// TIA Portal V20 export
// export: Created 2025-12-01T14:56:47.7137702Z, ExportSetting None, DisplayName Totally Integrated Automation Portal, DisplayVersion V20 Update 3, DisplayName TIA Portal Openness, DisplayVersion V20 Update 3, DisplayName TIA Portal Version Control Interface, DisplayVersion V20 Update 3, DisplayName STEP 7 Professional, DisplayVersion V20 Update 3, DisplayName STEP 7 Safety, DisplayVersion V20 Update 2, DisplayName WinCC Basic/Comfort/Advanced, DisplayVersion V20 Update 3, DisplayName WinCC Professional, DisplayVersion V20 Update 3, DisplayName WinCC Unified, DisplayVersion V20 Update 3
FUNCTION_BLOCK "FB350_Apilador_DesApilador_Paletas"   // FB350, LAD
TITLE = Control del Ramal de Salidas
{ S7_Optimized_Access := 'FALSE' }
AUTHOR : MAQUINA
NAME : 20181114
VERSION : 3.5
// Dani Palacios: Modificación octubre 2017 para poder desabilitar la maquina con un bit (por ejemplo en la puesta a punto si no esta montada o en el simulador)
// La modificación esta sin probar y es todo lo relativo a la variable Maquina_Desabilitada
// (bloqueo evolución desde etapa 0, bloqueo activación salidas en etapa 0 , fin vi sin mirar detectores y activación posición de reposo sin mirar detectores y variabkles de fin de movimiento).
// ES RESPONSABILIDAD DEL QUE DESABILITA LA MAQUINA QUE ESTA ESTE EN UNA POSICION QUE PERMITA EL MOVIMIENTO DE LAS CARGAS A TRAVES DE ELLA
// stored: AutoNumber false, SetENOAutomatically false
   VAR_INPUT
      Maquina : UInt;   // Numero de Maquina (Mesa)
      Error_Tx : Bool;   // Error en el Tx
      EnTension : Bool;   // Existe Tension en la Mesa
      MAQx_Desabilitada : Bool;   // Config MAQ. >>> DesHabilitada
      MAQx_ReposoDW : Bool;   // Config MAQ. >>> Pos. Reposo Abajo
      Termico_Elevacion : Bool;   // Termico de la Elevacion
      Termico_HorqDch : Bool;   // Termico de la Horquilla Derecha
      Termico_HorqIzq : Bool;   // Termico de la horquilla Izquierda
      pHsMx : Bool;   // pHs de la Mesa
      EnMovimiento_Tx : Bool;   // En Movimiento Tx
      pHs_LlenoApilador : Bool;   // Lleno el Apilador
      pHs_ConCargaApilador : Bool;   // ConCarga Apilador
      EM_UP : Bool;   // Emergencia Arriba del Apilador
      EM_DW : Bool;   // Emergencia Abajo del Apilador
      Pos_Dw : Bool;   // Posición Baja del Apilador
      Pos_Mid : Bool;   // Posición Media del Apilador
      Pos_Up : Bool;   // Posición Alta del Apilador
      Horq1_Der_Recogida : Bool;
      Horq2_Der_Recogida : Bool;
      Horq1_Izq_Recogida : Bool;
      Horq2_Izq_Recogida : Bool;
      Horq1_Der_Extendida : Bool;
      Horq2_Der_Extendida : Bool;
      Horq1_Izq_Extendida : Bool;
      Horq2_Izq_Extendida : Bool;
      EnMovimiento_Elevacion : Bool;   // En Movineto la Elevacion
      EnMovimiento_Horquillado : Bool;   // En Movimiento el Hoquillado
      PasarReposo_Apilador : Bool;   // Pasar a Reposo >>> Interlock Maquina
      CogerPila_Apilador : Bool;   // Coger la Pila >>> Interlock Maquina
      DispensarPaleta_Apilador : Bool;   // Dispensar Paleta >>> Interlock Maquina
      DispensarpPila_Apilador : Bool;   // Dispensar Pila >>> Interlock Maquina
      V_TIM_EstabilidadMov : Time := T#200MS;   // TIM de Estabilidad de los Mov.
      V_TOut_Elevacion : Int := 10000;   // TimeOut del Mov. de Elevacion
      V_TOut_Horquillado : Int := 3000;   // TimeOut del Mov. de Horquillado
   END_VAR
   VAR_OUTPUT
      Quieto_Apilador : Bool;   // Quieto >>> Interlock Maquina
      FinMovimiento_Apilador : Bool;   // Fin Movimiento >>> Interlock Maquina
   END_VAR
   VAR_IN_OUT
      StatusLleno_Apilador : Bool;   // Status Lleno >>> Interlock Maquina
      StatusSemiLleno_Apilador : Bool;   // Status SemiLleno >>> Interlock Maquina
      StatusVacio_Apilador : Bool;   // Status Vacio >>> Interlock Maquina
   END_VAR
   VAR
      Ap_ET00 : Bool;
      Ap_ET100 : Bool;
      Ap_ET101 : Bool;
      Ap_ET102 : Bool;
      Ap_ET103 : Bool;
      Ap_ET104 : Bool;
      Ap_ET105 : Bool;
      Ap_ET106 : Bool;
      Ap_ET107 : Bool;
      Ap_ET108 : Bool;
      Ap_ET109 : Bool;
      Ap_ET11 : Bool;
      Ap_ET12 : Bool;
      Ap_ET13 : Bool;
      Ap_ET14 : Bool;
      Ap_ET15 : Bool;
      Ap_ET16 : Bool;
      Ap_ET21 : Bool;
      Ap_ET22 : Bool;
      Ap_ET23 : Bool;
      Ap_ET24 : Bool;
      Ap_ET31 : Bool;
      Ap_ET32 : Bool;
      Ap_ET41 : Bool;
      Ap_ET42 : Bool;
      Ap_ET43 : Bool;
      Ap_ET44 : Bool;
      Ap_ET50 : Bool;
      Ap_ET51 : Bool;
      PosicionConocida : Bool;   // Interna >> Posicion Conocida
      Apilador_Lleno : Bool;   // Interna >> Lleno el Apilador
      HorquillasRecogidas : Bool;   // Carga Suelta en el Apilador
      HorquillasExtendidas : Bool;   // Carga Cogida en el Apilador
      STAT_FinMovimiento : Bool;   // Interna >> Fin Movimitnto del Apilador
      STAT_Quieto : Bool;   // Interna >> Quieto el Apilador
      CambioDir_SubidaBajada : Bool;   // Interna >> Cambio de Dir. Subida o Bajada
      MA_Ir_Up : Bool;   // ???
      MA_Ir_Dw : Bool;   // ???
      MA_Ir_Mid_Bajando : Bool;   // ???
      MA_Ir_Mid_Subiendo : Bool;   // ???
      MA_DejarCarga : Bool;   // ???
      MA_CogerCarga : Bool;   // ???
      TIM_EstabilidadMov { S7_SetPoint := 'True'} : TON_TIME;
      TMP_EnTension { S7_SetPoint := 'True'} : "FB910_CNT_UHS";
      TOut_Elevacion { S7_SetPoint := 'True'} : "FB910_CNT_UHS";
      TOut_Horquillado { S7_SetPoint := 'True'} : "FB910_CNT_UHS";
      Manual : "MoviManualMaquina_DesApilador";
   END_VAR
   VAR_TEMP
      EstadoZona : "EstadoZona";   // Estado de Zona de la Mesa
      EstadoMAQ : "EstadoMaquina_ApiladorDesapilador";   // Estado del Vehiculo Inteliguente de la Maquina
      Aux_ET00 : Bool;
   END_VAR
   VAR_TEMP   // added for the SCL form of the ladder/FBD networks
      _w1 : Bool;
   END_VAR
BEGIN

REGION Network 1: INICIALIZAR - Recoger las Variables de Estado de la Maquina
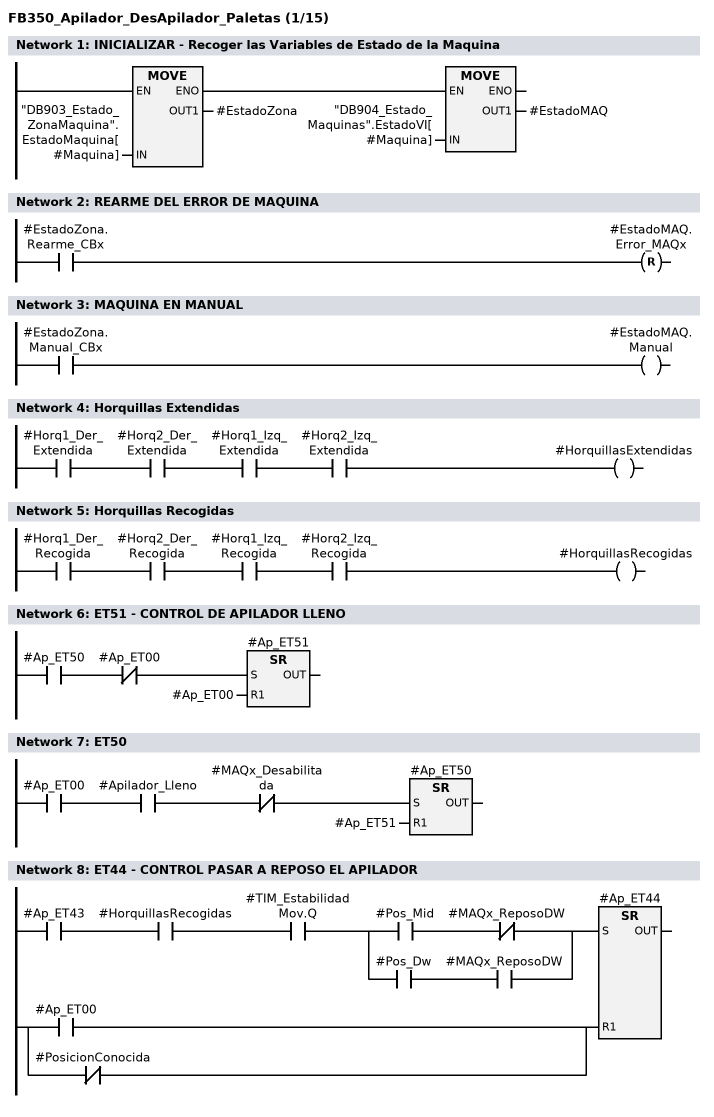
   RUNG wire#powerrail
      Move(in := "DB903_Estado_ZonaMaquina".EstadoMaquina[#Maquina], out1 => #EstadoZona)
      Move(in := "DB904_Estado_Maquinas".EstadoVI[#Maquina], out1 => #EstadoMAQ)
   END_RUNG
   // the same network as SCL:
   #EstadoZona := "DB903_Estado_ZonaMaquina".EstadoMaquina[#Maquina];
   #EstadoMAQ := "DB904_Estado_Maquinas".EstadoVI[#Maquina];
END_REGION

REGION Network 2: REARME DEL ERROR DE MAQUINA
   RUNG wire#powerrail
      Contact( #EstadoZona.Rearme_CBx )
      R_Coil( #EstadoMAQ.Error_MAQx )
   END_RUNG
   // the same network as SCL:
   IF #EstadoZona.Rearme_CBx THEN #EstadoMAQ.Error_MAQx := FALSE; END_IF;
END_REGION

REGION Network 3: MAQUINA EN MANUAL
   RUNG wire#powerrail
      Contact( #EstadoZona.Manual_CBx )
      Coil( #EstadoMAQ.Manual )
   END_RUNG
   // the same network as SCL:
   #EstadoMAQ.Manual := #EstadoZona.Manual_CBx;
END_REGION

REGION Network 4: Horquillas Extendidas
   RUNG wire#powerrail
      Contact( #Horq1_Der_Extendida )
      Contact( #Horq2_Der_Extendida )
      Contact( #Horq1_Izq_Extendida )
      Contact( #Horq2_Izq_Extendida )
      Coil( #HorquillasExtendidas )
   END_RUNG
   // the same network as SCL:
   #HorquillasExtendidas := #Horq1_Der_Extendida AND #Horq2_Der_Extendida AND #Horq1_Izq_Extendida AND #Horq2_Izq_Extendida;
END_REGION

REGION Network 5: Horquillas Recogidas
   RUNG wire#powerrail
      Contact( #Horq1_Der_Recogida )
      Contact( #Horq2_Der_Recogida )
      Contact( #Horq1_Izq_Recogida )
      Contact( #Horq2_Izq_Recogida )
      Coil( #HorquillasRecogidas )
   END_RUNG
   // the same network as SCL:
   #HorquillasRecogidas := #Horq1_Der_Recogida AND #Horq2_Der_Recogida AND #Horq1_Izq_Recogida AND #Horq2_Izq_Recogida;
END_REGION

REGION Network 6: ET51 - CONTROL DE APILADOR LLENO
   RUNG wire#powerrail
      Contact( #Ap_ET50 )
      I_Contact( #Ap_ET00 )
      S_SR(operand := #Ap_ET51, r1 := #Ap_ET00)
   END_RUNG
   // the same network as SCL:
   IF #Ap_ET50 AND NOT #Ap_ET00 THEN
       #Ap_ET51 := TRUE;   // SR flip-flop
   END_IF;
   IF #Ap_ET00 THEN #Ap_ET51 := FALSE; END_IF;
END_REGION

REGION Network 7: ET50
   RUNG wire#powerrail
      Contact( #Ap_ET00 )
      Contact( #Apilador_Lleno )
      I_Contact( #MAQx_Desabilitada )
      S_SR(operand := #Ap_ET50, r1 := #Ap_ET51)
   END_RUNG
   // the same network as SCL:
   IF #Ap_ET00 AND #Apilador_Lleno AND NOT #MAQx_Desabilitada THEN
       #Ap_ET50 := TRUE;   // SR flip-flop
   END_IF;
   IF #Ap_ET51 THEN #Ap_ET50 := FALSE; END_IF;
END_REGION

REGION Network 8: ET44 - CONTROL PASAR A REPOSO EL APILADOR
   RUNG wire#powerrail
      Contact( #Ap_ET43 )
      Contact( #HorquillasRecogidas )
      Contact( #TIM_EstabilidadMov.Q )
      wire#w1
      Contact( #Pos_Mid )
      I_Contact( #MAQx_ReposoDW )
      wire#w2
      S_SR(operand := #Ap_ET44, r1 := wire#w3)
   END_RUNG
   RUNG wire#w1
      Contact( #Pos_Dw )
      Contact( #MAQx_ReposoDW )
   END_RUNG wire#w2
   RUNG wire#powerrail
      Contact( #Ap_ET00 )
   END_RUNG wire#w3
   RUNG wire#powerrail
      I_Contact( #PosicionConocida )
   END_RUNG wire#w3
   // the same network as SCL:
   IF #Ap_ET43 AND #HorquillasRecogidas AND #TIM_EstabilidadMov.Q AND ((#Pos_Mid AND NOT #MAQx_ReposoDW) OR (#Pos_Dw AND #MAQx_ReposoDW)) THEN
       #Ap_ET44 := TRUE;   // SR flip-flop
   END_IF;
   IF #Ap_ET00 OR NOT #PosicionConocida THEN #Ap_ET44 := FALSE; END_IF;
END_REGION

REGION Network 9: ET43
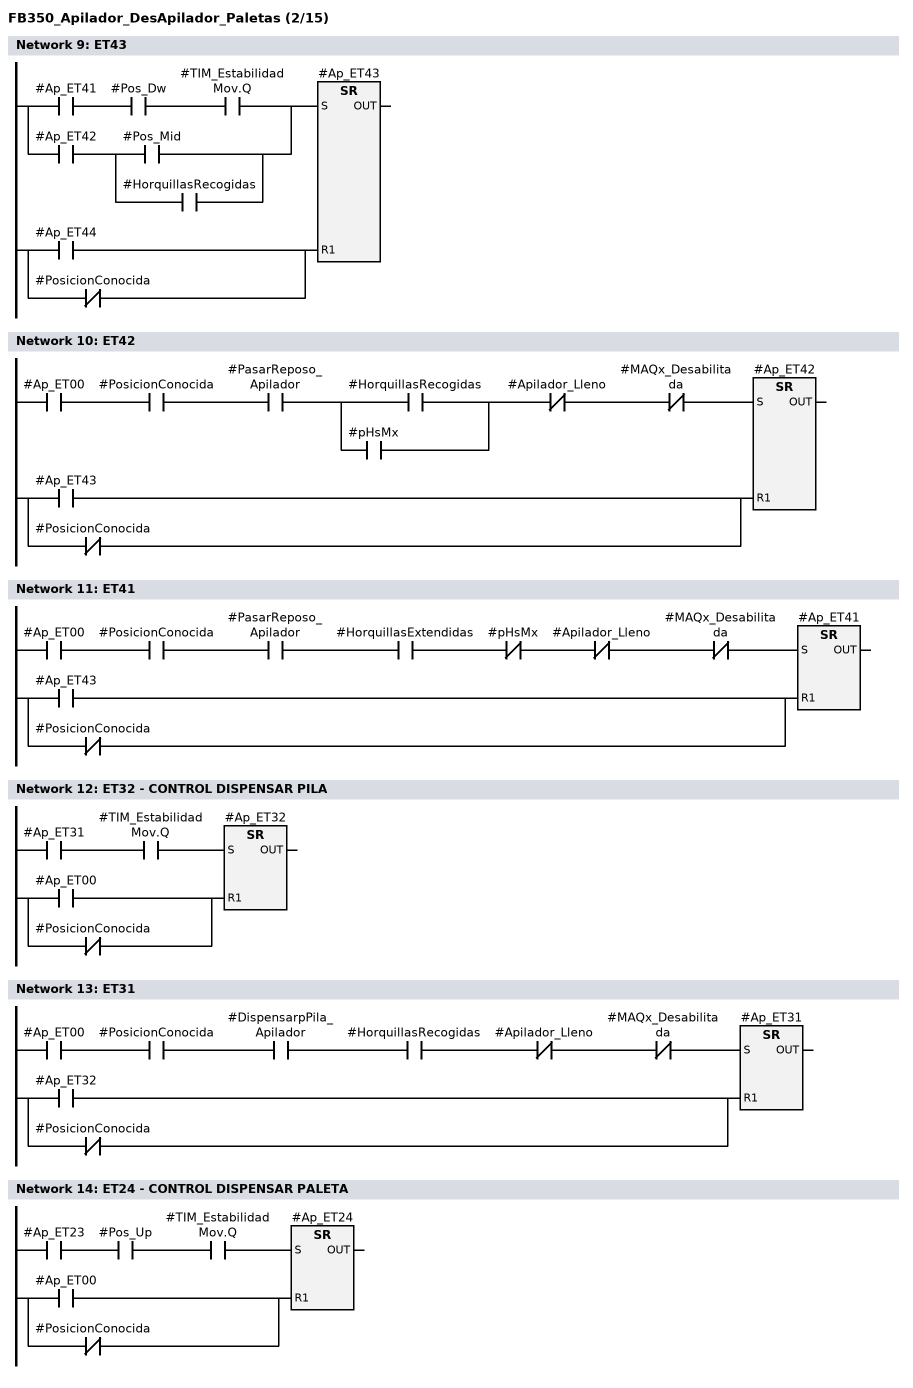
   RUNG wire#powerrail
      Contact( #Ap_ET41 )
      Contact( #Pos_Dw )
      Contact( #TIM_EstabilidadMov.Q )
      wire#w1
      S_SR(operand := #Ap_ET43, r1 := wire#w3)
   END_RUNG
   RUNG wire#powerrail
      Contact( #Ap_ET42 )
      wire#w2
      Contact( #Pos_Mid )
   END_RUNG wire#w1
   RUNG wire#w2
      Contact( #HorquillasRecogidas )
   END_RUNG wire#w1
   RUNG wire#powerrail
      Contact( #Ap_ET44 )
   END_RUNG wire#w3
   RUNG wire#powerrail
      I_Contact( #PosicionConocida )
   END_RUNG wire#w3
   // the same network as SCL:
   IF (#Ap_ET41 AND #Pos_Dw AND #TIM_EstabilidadMov.Q) OR (#Ap_ET42 AND (#Pos_Mid OR #HorquillasRecogidas)) THEN
       #Ap_ET43 := TRUE;   // SR flip-flop
   END_IF;
   IF #Ap_ET44 OR NOT #PosicionConocida THEN #Ap_ET43 := FALSE; END_IF;
END_REGION

REGION Network 10: ET42
   RUNG wire#powerrail
      Contact( #Ap_ET00 )
      Contact( #PosicionConocida )
      Contact( #PasarReposo_Apilador )
      wire#w1
      Contact( #HorquillasRecogidas )
      wire#w2
      I_Contact( #Apilador_Lleno )
      I_Contact( #MAQx_Desabilitada )
      S_SR(operand := #Ap_ET42, r1 := wire#w3)
   END_RUNG
   RUNG wire#w1
      Contact( #pHsMx )
   END_RUNG wire#w2
   RUNG wire#powerrail
      Contact( #Ap_ET43 )
   END_RUNG wire#w3
   RUNG wire#powerrail
      I_Contact( #PosicionConocida )
   END_RUNG wire#w3
   // the same network as SCL:
   IF #Ap_ET00 AND #PosicionConocida AND #PasarReposo_Apilador AND (#HorquillasRecogidas OR #pHsMx) AND NOT #Apilador_Lleno AND NOT #MAQx_Desabilitada THEN
       #Ap_ET42 := TRUE;   // SR flip-flop
   END_IF;
   IF #Ap_ET43 OR NOT #PosicionConocida THEN #Ap_ET42 := FALSE; END_IF;
END_REGION

REGION Network 11: ET41
   RUNG wire#powerrail
      Contact( #Ap_ET00 )
      Contact( #PosicionConocida )
      Contact( #PasarReposo_Apilador )
      Contact( #HorquillasExtendidas )
      I_Contact( #pHsMx )
      I_Contact( #Apilador_Lleno )
      I_Contact( #MAQx_Desabilitada )
      S_SR(operand := #Ap_ET41, r1 := wire#w1)
   END_RUNG
   RUNG wire#powerrail
      Contact( #Ap_ET43 )
   END_RUNG wire#w1
   RUNG wire#powerrail
      I_Contact( #PosicionConocida )
   END_RUNG wire#w1
   // the same network as SCL:
   IF #Ap_ET00 AND #PosicionConocida AND #PasarReposo_Apilador AND #HorquillasExtendidas AND NOT #pHsMx AND NOT #Apilador_Lleno AND NOT #MAQx_Desabilitada THEN
       #Ap_ET41 := TRUE;   // SR flip-flop
   END_IF;
   IF #Ap_ET43 OR NOT #PosicionConocida THEN #Ap_ET41 := FALSE; END_IF;
END_REGION

REGION Network 12: ET32 - CONTROL DISPENSAR PILA
   RUNG wire#powerrail
      Contact( #Ap_ET31 )
      Contact( #TIM_EstabilidadMov.Q )
      S_SR(operand := #Ap_ET32, r1 := wire#w1)
   END_RUNG
   RUNG wire#powerrail
      Contact( #Ap_ET00 )
   END_RUNG wire#w1
   RUNG wire#powerrail
      I_Contact( #PosicionConocida )
   END_RUNG wire#w1
   // the same network as SCL:
   IF #Ap_ET31 AND #TIM_EstabilidadMov.Q THEN
       #Ap_ET32 := TRUE;   // SR flip-flop
   END_IF;
   IF #Ap_ET00 OR NOT #PosicionConocida THEN #Ap_ET32 := FALSE; END_IF;
END_REGION

REGION Network 13: ET31
   RUNG wire#powerrail
      Contact( #Ap_ET00 )
      Contact( #PosicionConocida )
      Contact( #DispensarpPila_Apilador )
      Contact( #HorquillasRecogidas )
      I_Contact( #Apilador_Lleno )
      I_Contact( #MAQx_Desabilitada )
      S_SR(operand := #Ap_ET31, r1 := wire#w1)
   END_RUNG
   RUNG wire#powerrail
      Contact( #Ap_ET32 )
   END_RUNG wire#w1
   RUNG wire#powerrail
      I_Contact( #PosicionConocida )
   END_RUNG wire#w1
   // the same network as SCL:
   IF #Ap_ET00 AND #PosicionConocida AND #DispensarpPila_Apilador AND #HorquillasRecogidas AND NOT #Apilador_Lleno AND NOT #MAQx_Desabilitada THEN
       #Ap_ET31 := TRUE;   // SR flip-flop
   END_IF;
   IF #Ap_ET32 OR NOT #PosicionConocida THEN #Ap_ET31 := FALSE; END_IF;
END_REGION

REGION Network 14: ET24 - CONTROL DISPENSAR PALETA
   RUNG wire#powerrail
      Contact( #Ap_ET23 )
      Contact( #Pos_Up )
      Contact( #TIM_EstabilidadMov.Q )
      S_SR(operand := #Ap_ET24, r1 := wire#w1)
   END_RUNG
   RUNG wire#powerrail
      Contact( #Ap_ET00 )
   END_RUNG wire#w1
   RUNG wire#powerrail
      I_Contact( #PosicionConocida )
   END_RUNG wire#w1
   // the same network as SCL:
   IF #Ap_ET23 AND #Pos_Up AND #TIM_EstabilidadMov.Q THEN
       #Ap_ET24 := TRUE;   // SR flip-flop
   END_IF;
   IF #Ap_ET00 OR NOT #PosicionConocida THEN #Ap_ET24 := FALSE; END_IF;
END_REGION

REGION Network 15: ET23
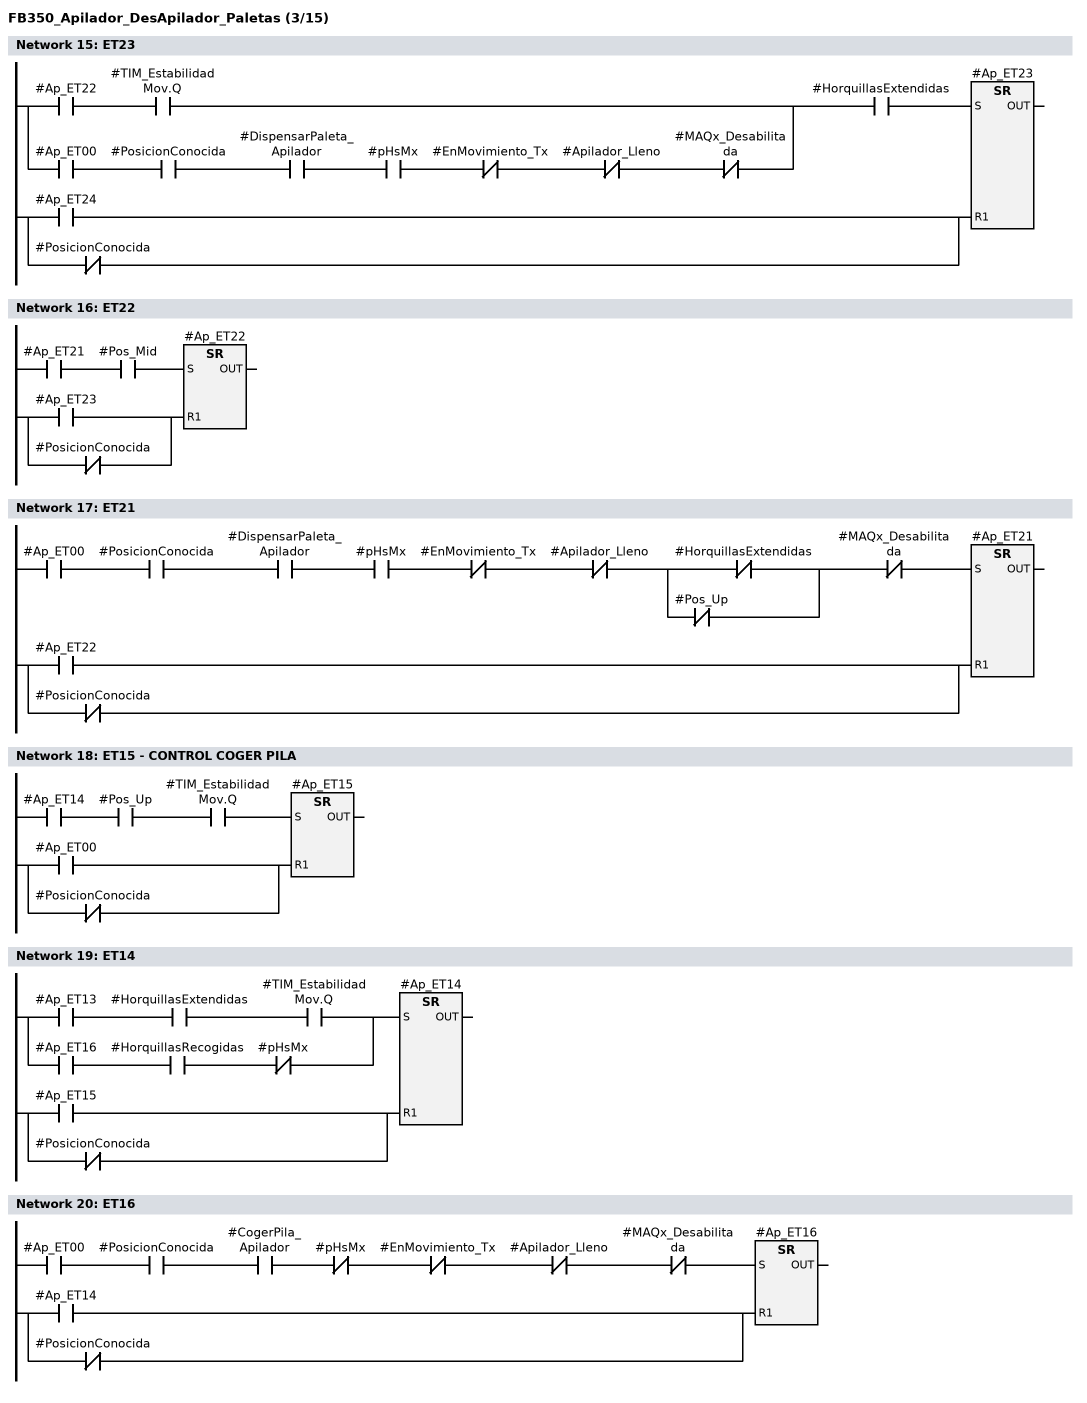
   RUNG wire#powerrail
      Contact( #Ap_ET22 )
      Contact( #TIM_EstabilidadMov.Q )
      wire#w1
      Contact( #HorquillasExtendidas )
      S_SR(operand := #Ap_ET23, r1 := wire#w2)
   END_RUNG
   RUNG wire#powerrail
      Contact( #Ap_ET00 )
      Contact( #PosicionConocida )
      Contact( #DispensarPaleta_Apilador )
      Contact( #pHsMx )
      I_Contact( #EnMovimiento_Tx )
      I_Contact( #Apilador_Lleno )
      I_Contact( #MAQx_Desabilitada )
   END_RUNG wire#w1
   RUNG wire#powerrail
      Contact( #Ap_ET24 )
   END_RUNG wire#w2
   RUNG wire#powerrail
      I_Contact( #PosicionConocida )
   END_RUNG wire#w2
   // the same network as SCL:
   IF ((#Ap_ET22 AND #TIM_EstabilidadMov.Q) OR (#Ap_ET00 AND #PosicionConocida AND #DispensarPaleta_Apilador AND #pHsMx AND NOT #EnMovimiento_Tx AND NOT #Apilador_Lleno AND NOT #MAQx_Desabilitada)) AND #HorquillasExtendidas THEN
       #Ap_ET23 := TRUE;   // SR flip-flop
   END_IF;
   IF #Ap_ET24 OR NOT #PosicionConocida THEN #Ap_ET23 := FALSE; END_IF;
END_REGION

REGION Network 16: ET22
   RUNG wire#powerrail
      Contact( #Ap_ET21 )
      Contact( #Pos_Mid )
      S_SR(operand := #Ap_ET22, r1 := wire#w1)
   END_RUNG
   RUNG wire#powerrail
      Contact( #Ap_ET23 )
   END_RUNG wire#w1
   RUNG wire#powerrail
      I_Contact( #PosicionConocida )
   END_RUNG wire#w1
   // the same network as SCL:
   IF #Ap_ET21 AND #Pos_Mid THEN
       #Ap_ET22 := TRUE;   // SR flip-flop
   END_IF;
   IF #Ap_ET23 OR NOT #PosicionConocida THEN #Ap_ET22 := FALSE; END_IF;
END_REGION

REGION Network 17: ET21
   RUNG wire#powerrail
      Contact( #Ap_ET00 )
      Contact( #PosicionConocida )
      Contact( #DispensarPaleta_Apilador )
      Contact( #pHsMx )
      I_Contact( #EnMovimiento_Tx )
      I_Contact( #Apilador_Lleno )
      wire#w1
      I_Contact( #HorquillasExtendidas )
      wire#w2
      I_Contact( #MAQx_Desabilitada )
      S_SR(operand := #Ap_ET21, r1 := wire#w3)
   END_RUNG
   RUNG wire#w1
      I_Contact( #Pos_Up )
   END_RUNG wire#w2
   RUNG wire#powerrail
      Contact( #Ap_ET22 )
   END_RUNG wire#w3
   RUNG wire#powerrail
      I_Contact( #PosicionConocida )
   END_RUNG wire#w3
   // the same network as SCL:
   IF #Ap_ET00 AND #PosicionConocida AND #DispensarPaleta_Apilador AND #pHsMx AND NOT #EnMovimiento_Tx AND NOT #Apilador_Lleno AND (NOT #HorquillasExtendidas OR NOT #Pos_Up) AND NOT #MAQx_Desabilitada THEN
       #Ap_ET21 := TRUE;   // SR flip-flop
   END_IF;
   IF #Ap_ET22 OR NOT #PosicionConocida THEN #Ap_ET21 := FALSE; END_IF;
END_REGION

REGION Network 18: ET15 - CONTROL COGER PILA
   RUNG wire#powerrail
      Contact( #Ap_ET14 )
      Contact( #Pos_Up )
      Contact( #TIM_EstabilidadMov.Q )
      S_SR(operand := #Ap_ET15, r1 := wire#w1)
   END_RUNG
   RUNG wire#powerrail
      Contact( #Ap_ET00 )
   END_RUNG wire#w1
   RUNG wire#powerrail
      I_Contact( #PosicionConocida )
   END_RUNG wire#w1
   // the same network as SCL:
   IF #Ap_ET14 AND #Pos_Up AND #TIM_EstabilidadMov.Q THEN
       #Ap_ET15 := TRUE;   // SR flip-flop
   END_IF;
   IF #Ap_ET00 OR NOT #PosicionConocida THEN #Ap_ET15 := FALSE; END_IF;
END_REGION

REGION Network 19: ET14
   RUNG wire#powerrail
      Contact( #Ap_ET13 )
      Contact( #HorquillasExtendidas )
      Contact( #TIM_EstabilidadMov.Q )
      wire#w1
      S_SR(operand := #Ap_ET14, r1 := wire#w2)
   END_RUNG
   RUNG wire#powerrail
      Contact( #Ap_ET16 )
      Contact( #HorquillasRecogidas )
      I_Contact( #pHsMx )
   END_RUNG wire#w1
   RUNG wire#powerrail
      Contact( #Ap_ET15 )
   END_RUNG wire#w2
   RUNG wire#powerrail
      I_Contact( #PosicionConocida )
   END_RUNG wire#w2
   // the same network as SCL:
   IF (#Ap_ET13 AND #HorquillasExtendidas AND #TIM_EstabilidadMov.Q) OR (#Ap_ET16 AND #HorquillasRecogidas AND NOT #pHsMx) THEN
       #Ap_ET14 := TRUE;   // SR flip-flop
   END_IF;
   IF #Ap_ET15 OR NOT #PosicionConocida THEN #Ap_ET14 := FALSE; END_IF;
END_REGION

REGION Network 20: ET16
   RUNG wire#powerrail
      Contact( #Ap_ET00 )
      Contact( #PosicionConocida )
      Contact( #CogerPila_Apilador )
      I_Contact( #pHsMx )
      I_Contact( #EnMovimiento_Tx )
      I_Contact( #Apilador_Lleno )
      I_Contact( #MAQx_Desabilitada )
      S_SR(operand := #Ap_ET16, r1 := wire#w1)
   END_RUNG
   RUNG wire#powerrail
      Contact( #Ap_ET14 )
   END_RUNG wire#w1
   RUNG wire#powerrail
      I_Contact( #PosicionConocida )
   END_RUNG wire#w1
   // the same network as SCL:
   IF #Ap_ET00 AND #PosicionConocida AND #CogerPila_Apilador AND NOT #pHsMx AND NOT #EnMovimiento_Tx AND NOT #Apilador_Lleno AND NOT #MAQx_Desabilitada THEN
       #Ap_ET16 := TRUE;   // SR flip-flop
   END_IF;
   IF #Ap_ET14 OR NOT #PosicionConocida THEN #Ap_ET16 := FALSE; END_IF;
END_REGION

REGION Network 21: ET13
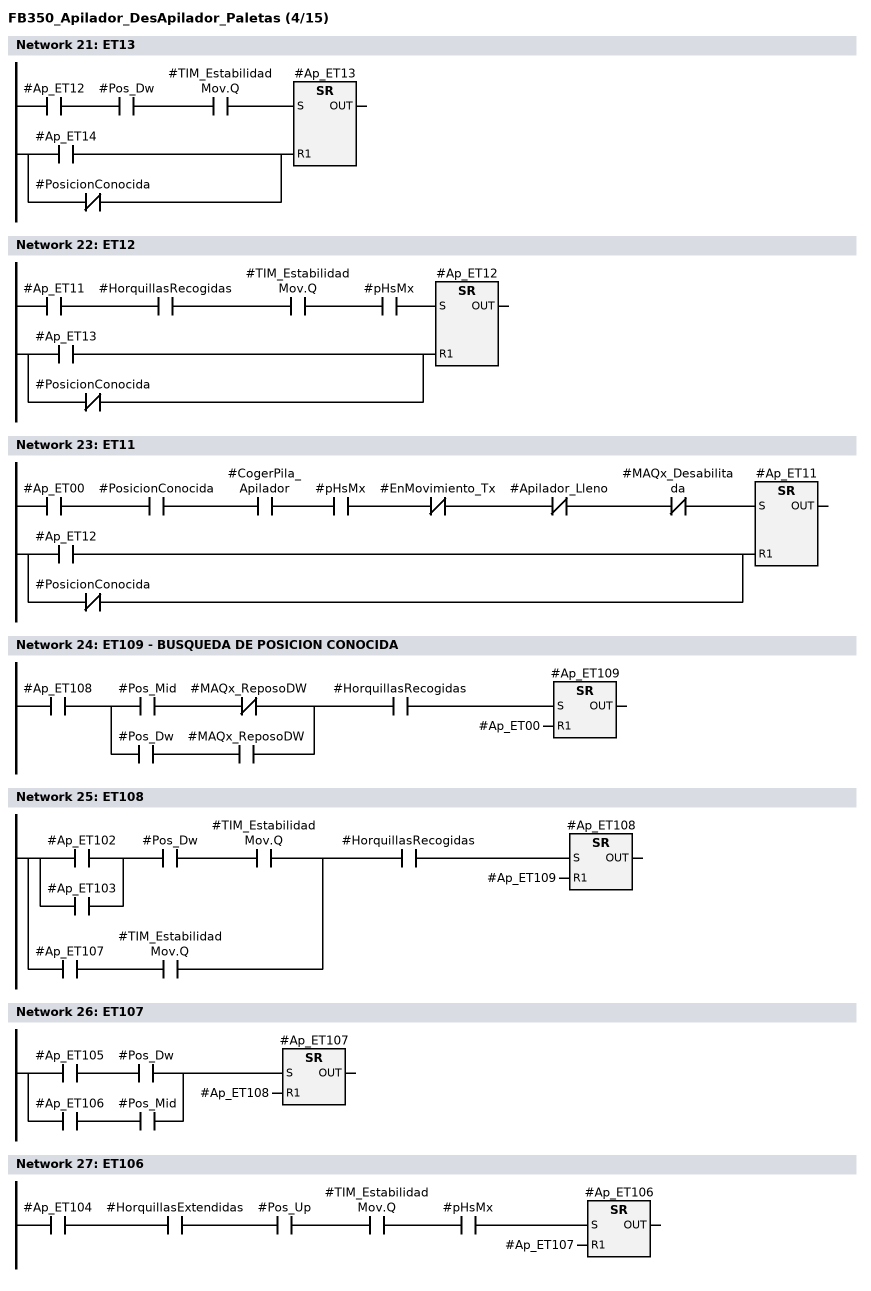
   RUNG wire#powerrail
      Contact( #Ap_ET12 )
      Contact( #Pos_Dw )
      Contact( #TIM_EstabilidadMov.Q )
      S_SR(operand := #Ap_ET13, r1 := wire#w1)
   END_RUNG
   RUNG wire#powerrail
      Contact( #Ap_ET14 )
   END_RUNG wire#w1
   RUNG wire#powerrail
      I_Contact( #PosicionConocida )
   END_RUNG wire#w1
   // the same network as SCL:
   IF #Ap_ET12 AND #Pos_Dw AND #TIM_EstabilidadMov.Q THEN
       #Ap_ET13 := TRUE;   // SR flip-flop
   END_IF;
   IF #Ap_ET14 OR NOT #PosicionConocida THEN #Ap_ET13 := FALSE; END_IF;
END_REGION

REGION Network 22: ET12
   RUNG wire#powerrail
      Contact( #Ap_ET11 )
      Contact( #HorquillasRecogidas )
      Contact( #TIM_EstabilidadMov.Q )
      Contact( #pHsMx )
      S_SR(operand := #Ap_ET12, r1 := wire#w1)
   END_RUNG
   RUNG wire#powerrail
      Contact( #Ap_ET13 )
   END_RUNG wire#w1
   RUNG wire#powerrail
      I_Contact( #PosicionConocida )
   END_RUNG wire#w1
   // the same network as SCL:
   IF #Ap_ET11 AND #HorquillasRecogidas AND #TIM_EstabilidadMov.Q AND #pHsMx THEN
       #Ap_ET12 := TRUE;   // SR flip-flop
   END_IF;
   IF #Ap_ET13 OR NOT #PosicionConocida THEN #Ap_ET12 := FALSE; END_IF;
END_REGION

REGION Network 23: ET11
   RUNG wire#powerrail
      Contact( #Ap_ET00 )
      Contact( #PosicionConocida )
      Contact( #CogerPila_Apilador )
      Contact( #pHsMx )
      I_Contact( #EnMovimiento_Tx )
      I_Contact( #Apilador_Lleno )
      I_Contact( #MAQx_Desabilitada )
      S_SR(operand := #Ap_ET11, r1 := wire#w1)
   END_RUNG
   RUNG wire#powerrail
      Contact( #Ap_ET12 )
   END_RUNG wire#w1
   RUNG wire#powerrail
      I_Contact( #PosicionConocida )
   END_RUNG wire#w1
   // the same network as SCL:
   IF #Ap_ET00 AND #PosicionConocida AND #CogerPila_Apilador AND #pHsMx AND NOT #EnMovimiento_Tx AND NOT #Apilador_Lleno AND NOT #MAQx_Desabilitada THEN
       #Ap_ET11 := TRUE;   // SR flip-flop
   END_IF;
   IF #Ap_ET12 OR NOT #PosicionConocida THEN #Ap_ET11 := FALSE; END_IF;
END_REGION

REGION Network 24: ET109 - BUSQUEDA DE POSICION CONOCIDA
   RUNG wire#powerrail
      Contact( #Ap_ET108 )
      wire#w1
      Contact( #Pos_Mid )
      I_Contact( #MAQx_ReposoDW )
      wire#w2
      Contact( #HorquillasRecogidas )
      S_SR(operand := #Ap_ET109, r1 := #Ap_ET00)
   END_RUNG
   RUNG wire#w1
      Contact( #Pos_Dw )
      Contact( #MAQx_ReposoDW )
   END_RUNG wire#w2
   // the same network as SCL:
   IF #Ap_ET108 AND ((#Pos_Mid AND NOT #MAQx_ReposoDW) OR (#Pos_Dw AND #MAQx_ReposoDW)) AND #HorquillasRecogidas THEN
       #Ap_ET109 := TRUE;   // SR flip-flop
   END_IF;
   IF #Ap_ET00 THEN #Ap_ET109 := FALSE; END_IF;
END_REGION

REGION Network 25: ET108
   RUNG wire#powerrail
      Contact( #Ap_ET102 )
      wire#w1
      Contact( #Pos_Dw )
      Contact( #TIM_EstabilidadMov.Q )
      wire#w2
      Contact( #HorquillasRecogidas )
      S_SR(operand := #Ap_ET108, r1 := #Ap_ET109)
   END_RUNG
   RUNG wire#powerrail
      Contact( #Ap_ET103 )
   END_RUNG wire#w1
   RUNG wire#powerrail
      Contact( #Ap_ET107 )
      Contact( #TIM_EstabilidadMov.Q )
   END_RUNG wire#w2
   // the same network as SCL:
   IF (((#Ap_ET102 OR #Ap_ET103) AND #Pos_Dw AND #TIM_EstabilidadMov.Q) OR (#Ap_ET107 AND #TIM_EstabilidadMov.Q)) AND #HorquillasRecogidas THEN
       #Ap_ET108 := TRUE;   // SR flip-flop
   END_IF;
   IF #Ap_ET109 THEN #Ap_ET108 := FALSE; END_IF;
END_REGION

REGION Network 26: ET107
   RUNG wire#powerrail
      Contact( #Ap_ET105 )
      Contact( #Pos_Dw )
      wire#w1
      S_SR(operand := #Ap_ET107, r1 := #Ap_ET108)
   END_RUNG
   RUNG wire#powerrail
      Contact( #Ap_ET106 )
      Contact( #Pos_Mid )
   END_RUNG wire#w1
   // the same network as SCL:
   IF (#Ap_ET105 AND #Pos_Dw) OR (#Ap_ET106 AND #Pos_Mid) THEN
       #Ap_ET107 := TRUE;   // SR flip-flop
   END_IF;
   IF #Ap_ET108 THEN #Ap_ET107 := FALSE; END_IF;
END_REGION

REGION Network 27: ET106
   RUNG wire#powerrail
      Contact( #Ap_ET104 )
      Contact( #HorquillasExtendidas )
      Contact( #Pos_Up )
      Contact( #TIM_EstabilidadMov.Q )
      Contact( #pHsMx )
      S_SR(operand := #Ap_ET106, r1 := #Ap_ET107)
   END_RUNG
   // the same network as SCL:
   IF #Ap_ET104 AND #HorquillasExtendidas AND #Pos_Up AND #TIM_EstabilidadMov.Q AND #pHsMx THEN
       #Ap_ET106 := TRUE;   // SR flip-flop
   END_IF;
   IF #Ap_ET107 THEN #Ap_ET106 := FALSE; END_IF;
END_REGION

REGION Network 28: ET105
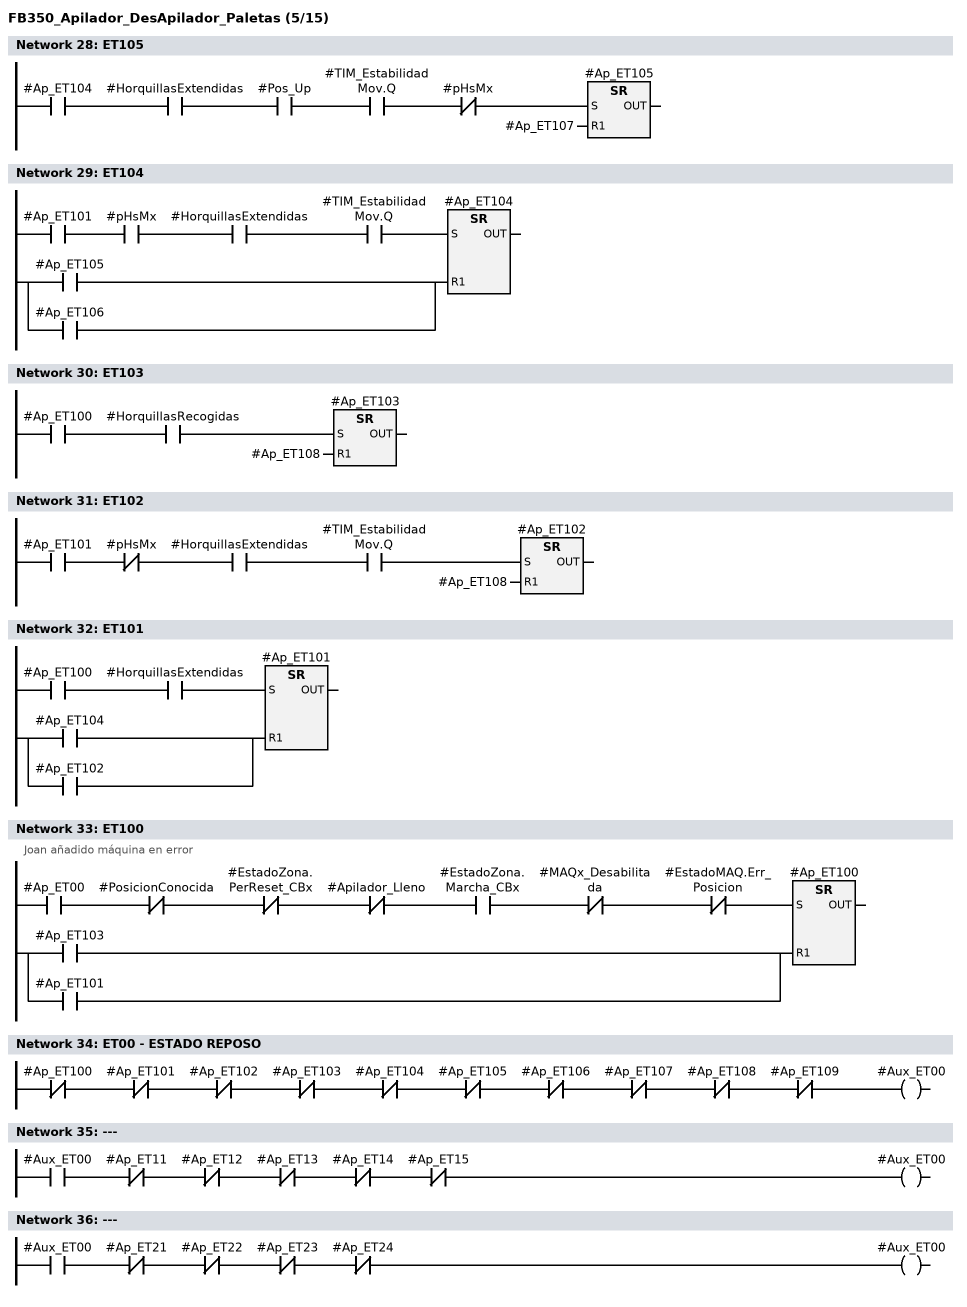
   RUNG wire#powerrail
      Contact( #Ap_ET104 )
      Contact( #HorquillasExtendidas )
      Contact( #Pos_Up )
      Contact( #TIM_EstabilidadMov.Q )
      I_Contact( #pHsMx )
      S_SR(operand := #Ap_ET105, r1 := #Ap_ET107)
   END_RUNG
   // the same network as SCL:
   IF #Ap_ET104 AND #HorquillasExtendidas AND #Pos_Up AND #TIM_EstabilidadMov.Q AND NOT #pHsMx THEN
       #Ap_ET105 := TRUE;   // SR flip-flop
   END_IF;
   IF #Ap_ET107 THEN #Ap_ET105 := FALSE; END_IF;
END_REGION

REGION Network 29: ET104
   RUNG wire#powerrail
      Contact( #Ap_ET101 )
      Contact( #pHsMx )
      Contact( #HorquillasExtendidas )
      Contact( #TIM_EstabilidadMov.Q )
      S_SR(operand := #Ap_ET104, r1 := wire#w1)
   END_RUNG
   RUNG wire#powerrail
      Contact( #Ap_ET105 )
   END_RUNG wire#w1
   RUNG wire#powerrail
      Contact( #Ap_ET106 )
   END_RUNG wire#w1
   // the same network as SCL:
   IF #Ap_ET101 AND #pHsMx AND #HorquillasExtendidas AND #TIM_EstabilidadMov.Q THEN
       #Ap_ET104 := TRUE;   // SR flip-flop
   END_IF;
   IF #Ap_ET105 OR #Ap_ET106 THEN #Ap_ET104 := FALSE; END_IF;
END_REGION

REGION Network 30: ET103
   RUNG wire#powerrail
      Contact( #Ap_ET100 )
      Contact( #HorquillasRecogidas )
      S_SR(operand := #Ap_ET103, r1 := #Ap_ET108)
   END_RUNG
   // the same network as SCL:
   IF #Ap_ET100 AND #HorquillasRecogidas THEN
       #Ap_ET103 := TRUE;   // SR flip-flop
   END_IF;
   IF #Ap_ET108 THEN #Ap_ET103 := FALSE; END_IF;
END_REGION

REGION Network 31: ET102
   RUNG wire#powerrail
      Contact( #Ap_ET101 )
      I_Contact( #pHsMx )
      Contact( #HorquillasExtendidas )
      Contact( #TIM_EstabilidadMov.Q )
      S_SR(operand := #Ap_ET102, r1 := #Ap_ET108)
   END_RUNG
   // the same network as SCL:
   IF #Ap_ET101 AND NOT #pHsMx AND #HorquillasExtendidas AND #TIM_EstabilidadMov.Q THEN
       #Ap_ET102 := TRUE;   // SR flip-flop
   END_IF;
   IF #Ap_ET108 THEN #Ap_ET102 := FALSE; END_IF;
END_REGION

REGION Network 32: ET101
   RUNG wire#powerrail
      Contact( #Ap_ET100 )
      Contact( #HorquillasExtendidas )
      S_SR(operand := #Ap_ET101, r1 := wire#w1)
   END_RUNG
   RUNG wire#powerrail
      Contact( #Ap_ET104 )
   END_RUNG wire#w1
   RUNG wire#powerrail
      Contact( #Ap_ET102 )
   END_RUNG wire#w1
   // the same network as SCL:
   IF #Ap_ET100 AND #HorquillasExtendidas THEN
       #Ap_ET101 := TRUE;   // SR flip-flop
   END_IF;
   IF #Ap_ET104 OR #Ap_ET102 THEN #Ap_ET101 := FALSE; END_IF;
END_REGION

REGION Network 33: ET100
   // Joan añadido máquina en error
   RUNG wire#powerrail
      Contact( #Ap_ET00 )
      I_Contact( #PosicionConocida )
      I_Contact( #EstadoZona.PerReset_CBx )
      I_Contact( #Apilador_Lleno )
      Contact( #EstadoZona.Marcha_CBx )
      I_Contact( #MAQx_Desabilitada )
      I_Contact( #EstadoMAQ.Err_Posicion )
      S_SR(operand := #Ap_ET100, r1 := wire#w1)
   END_RUNG
   RUNG wire#powerrail
      Contact( #Ap_ET103 )
   END_RUNG wire#w1
   RUNG wire#powerrail
      Contact( #Ap_ET101 )
   END_RUNG wire#w1
   // the same network as SCL:
   IF #Ap_ET00 AND NOT #PosicionConocida AND NOT #EstadoZona.PerReset_CBx AND NOT #Apilador_Lleno AND #EstadoZona.Marcha_CBx AND NOT #MAQx_Desabilitada AND NOT #EstadoMAQ.Err_Posicion THEN
       #Ap_ET100 := TRUE;   // SR flip-flop
   END_IF;
   IF #Ap_ET103 OR #Ap_ET101 THEN #Ap_ET100 := FALSE; END_IF;
END_REGION

REGION Network 34: ET00 - ESTADO REPOSO
   RUNG wire#powerrail
      I_Contact( #Ap_ET100 )
      I_Contact( #Ap_ET101 )
      I_Contact( #Ap_ET102 )
      I_Contact( #Ap_ET103 )
      I_Contact( #Ap_ET104 )
      I_Contact( #Ap_ET105 )
      I_Contact( #Ap_ET106 )
      I_Contact( #Ap_ET107 )
      I_Contact( #Ap_ET108 )
      I_Contact( #Ap_ET109 )
      Coil( #Aux_ET00 )
   END_RUNG
   // the same network as SCL:
   #Aux_ET00 := NOT #Ap_ET100 AND NOT #Ap_ET101 AND NOT #Ap_ET102 AND NOT #Ap_ET103 AND NOT #Ap_ET104 AND NOT #Ap_ET105 AND NOT #Ap_ET106 AND NOT #Ap_ET107 AND NOT #Ap_ET108 AND NOT #Ap_ET109;
END_REGION

REGION Network 35: ---
   RUNG wire#powerrail
      Contact( #Aux_ET00 )
      I_Contact( #Ap_ET11 )
      I_Contact( #Ap_ET12 )
      I_Contact( #Ap_ET13 )
      I_Contact( #Ap_ET14 )
      I_Contact( #Ap_ET15 )
      Coil( #Aux_ET00 )
   END_RUNG
   // the same network as SCL:
   #Aux_ET00 := #Aux_ET00 AND NOT #Ap_ET11 AND NOT #Ap_ET12 AND NOT #Ap_ET13 AND NOT #Ap_ET14 AND NOT #Ap_ET15;
END_REGION

REGION Network 36: ---
   RUNG wire#powerrail
      Contact( #Aux_ET00 )
      I_Contact( #Ap_ET21 )
      I_Contact( #Ap_ET22 )
      I_Contact( #Ap_ET23 )
      I_Contact( #Ap_ET24 )
      Coil( #Aux_ET00 )
   END_RUNG
   // the same network as SCL:
   #Aux_ET00 := #Aux_ET00 AND NOT #Ap_ET21 AND NOT #Ap_ET22 AND NOT #Ap_ET23 AND NOT #Ap_ET24;
END_REGION

REGION Network 37: ---
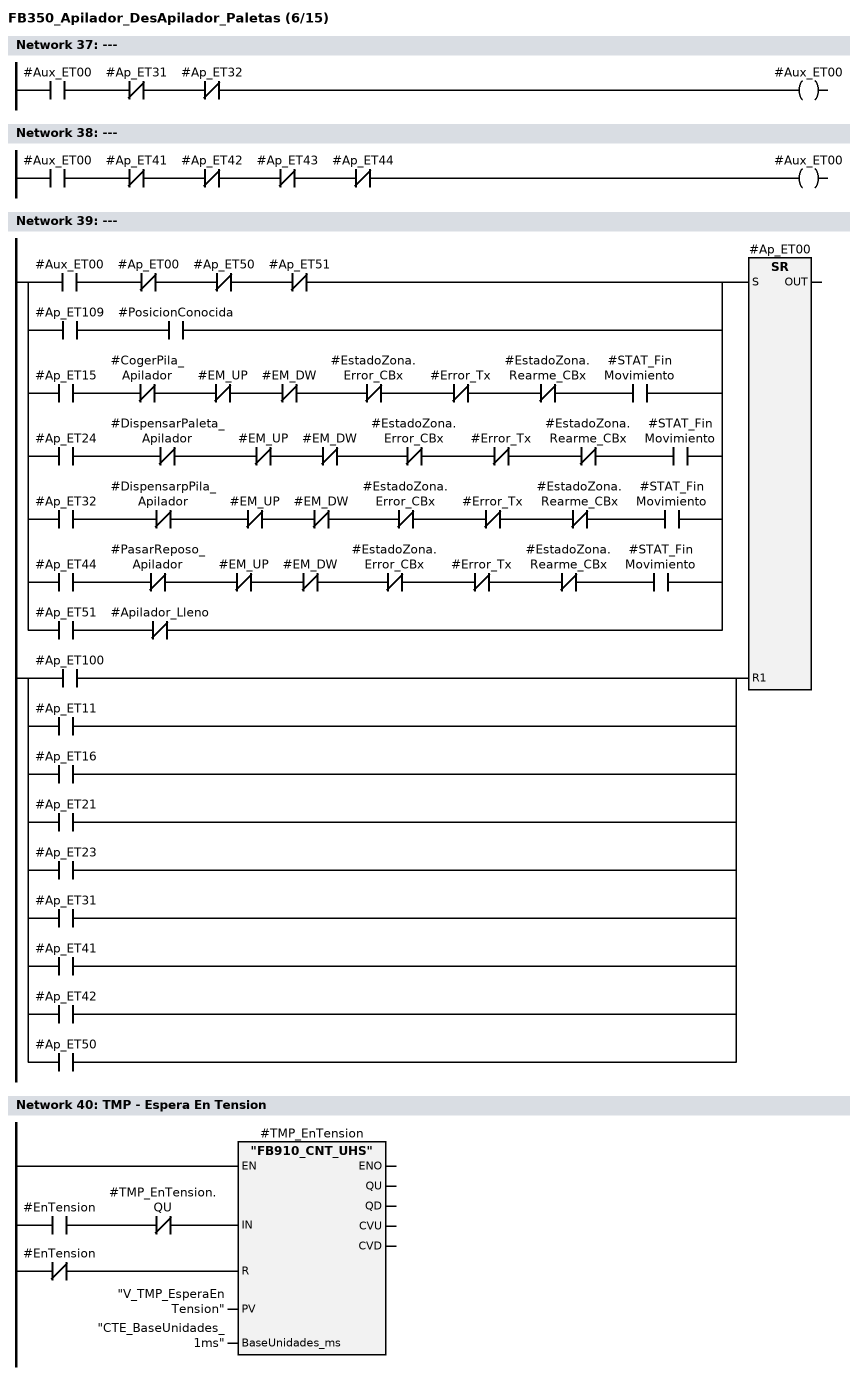
   RUNG wire#powerrail
      Contact( #Aux_ET00 )
      I_Contact( #Ap_ET31 )
      I_Contact( #Ap_ET32 )
      Coil( #Aux_ET00 )
   END_RUNG
   // the same network as SCL:
   #Aux_ET00 := #Aux_ET00 AND NOT #Ap_ET31 AND NOT #Ap_ET32;
END_REGION

REGION Network 38: ---
   RUNG wire#powerrail
      Contact( #Aux_ET00 )
      I_Contact( #Ap_ET41 )
      I_Contact( #Ap_ET42 )
      I_Contact( #Ap_ET43 )
      I_Contact( #Ap_ET44 )
      Coil( #Aux_ET00 )
   END_RUNG
   // the same network as SCL:
   #Aux_ET00 := #Aux_ET00 AND NOT #Ap_ET41 AND NOT #Ap_ET42 AND NOT #Ap_ET43 AND NOT #Ap_ET44;
END_REGION

REGION Network 39: ---
   RUNG wire#powerrail
      Contact( #Aux_ET00 )
      I_Contact( #Ap_ET00 )
      I_Contact( #Ap_ET50 )
      I_Contact( #Ap_ET51 )
      wire#w1
      S_SR(operand := #Ap_ET00, r1 := wire#w2)
   END_RUNG
   RUNG wire#powerrail
      Contact( #Ap_ET109 )
      Contact( #PosicionConocida )
   END_RUNG wire#w1
   RUNG wire#powerrail
      Contact( #Ap_ET15 )
      I_Contact( #CogerPila_Apilador )
      I_Contact( #EM_UP )
      I_Contact( #EM_DW )
      I_Contact( #EstadoZona.Error_CBx )
      I_Contact( #Error_Tx )
      I_Contact( #EstadoZona.Rearme_CBx )
      Contact( #STAT_FinMovimiento )
   END_RUNG wire#w1
   RUNG wire#powerrail
      Contact( #Ap_ET24 )
      I_Contact( #DispensarPaleta_Apilador )
      I_Contact( #EM_UP )
      I_Contact( #EM_DW )
      I_Contact( #EstadoZona.Error_CBx )
      I_Contact( #Error_Tx )
      I_Contact( #EstadoZona.Rearme_CBx )
      Contact( #STAT_FinMovimiento )
   END_RUNG wire#w1
   RUNG wire#powerrail
      Contact( #Ap_ET32 )
      I_Contact( #DispensarpPila_Apilador )
      I_Contact( #EM_UP )
      I_Contact( #EM_DW )
      I_Contact( #EstadoZona.Error_CBx )
      I_Contact( #Error_Tx )
      I_Contact( #EstadoZona.Rearme_CBx )
      Contact( #STAT_FinMovimiento )
   END_RUNG wire#w1
   RUNG wire#powerrail
      Contact( #Ap_ET44 )
      I_Contact( #PasarReposo_Apilador )
      I_Contact( #EM_UP )
      I_Contact( #EM_DW )
      I_Contact( #EstadoZona.Error_CBx )
      I_Contact( #Error_Tx )
      I_Contact( #EstadoZona.Rearme_CBx )
      Contact( #STAT_FinMovimiento )
   END_RUNG wire#w1
   RUNG wire#powerrail
      Contact( #Ap_ET51 )
      I_Contact( #Apilador_Lleno )
   END_RUNG wire#w1
   RUNG wire#powerrail
      Contact( #Ap_ET100 )
   END_RUNG wire#w2
   RUNG wire#powerrail
      Contact( #Ap_ET11 )
   END_RUNG wire#w2
   RUNG wire#powerrail
      Contact( #Ap_ET16 )
   END_RUNG wire#w2
   RUNG wire#powerrail
      Contact( #Ap_ET21 )
   END_RUNG wire#w2
   RUNG wire#powerrail
      Contact( #Ap_ET23 )
   END_RUNG wire#w2
   RUNG wire#powerrail
      Contact( #Ap_ET31 )
   END_RUNG wire#w2
   RUNG wire#powerrail
      Contact( #Ap_ET41 )
   END_RUNG wire#w2
   RUNG wire#powerrail
      Contact( #Ap_ET42 )
   END_RUNG wire#w2
   RUNG wire#powerrail
      Contact( #Ap_ET50 )
   END_RUNG wire#w2
   // the same network as SCL:
   IF (#Aux_ET00 AND NOT #Ap_ET00 AND NOT #Ap_ET50 AND NOT #Ap_ET51) OR (#Ap_ET109 AND #PosicionConocida) OR (#Ap_ET15 AND NOT #CogerPila_Apilador AND NOT #EM_UP AND NOT #EM_DW AND NOT #EstadoZona.Error_CBx AND NOT #Error_Tx AND NOT #EstadoZona.Rearme_CBx AND #STAT_FinMovimiento) OR (#Ap_ET24 AND NOT #DispensarPaleta_Apilador AND NOT #EM_UP AND NOT #EM_DW AND NOT #EstadoZona.Error_CBx AND NOT #Error_Tx AND NOT #EstadoZona.Rearme_CBx AND #STAT_FinMovimiento) OR (#Ap_ET32 AND NOT #DispensarpPila_Apilador AND NOT #EM_UP AND NOT #EM_DW AND NOT #EstadoZona.Error_CBx AND NOT #Error_Tx AND NOT #EstadoZona.Rearme_CBx AND #STAT_FinMovimiento) OR (#Ap_ET44 AND NOT #PasarReposo_Apilador AND NOT #EM_UP AND NOT #EM_DW AND NOT #EstadoZona.Error_CBx AND NOT #Error_Tx AND NOT #EstadoZona.Rearme_CBx AND #STAT_FinMovimiento) OR (#Ap_ET51 AND NOT #Apilador_Lleno) THEN
       #Ap_ET00 := TRUE;   // SR flip-flop
   END_IF;
   IF #Ap_ET100 OR #Ap_ET11 OR #Ap_ET16 OR #Ap_ET21 OR #Ap_ET23 OR #Ap_ET31 OR #Ap_ET41 OR #Ap_ET42 OR #Ap_ET50 THEN
       #Ap_ET00 := FALSE;
   END_IF;
END_REGION

REGION Network 40: TMP - Espera En Tension
   RUNG wire#powerrail
      #TMP_EnTension(IN := wire#w1, R := wire#w2, PV := "V_TMP_EsperaEnTension", BaseUnidades_ms := "CTE_BaseUnidades_1ms", QU =>, QD =>, CVU =>, CVD =>)
   END_RUNG
   RUNG wire#powerrail
      Contact( #EnTension )
      I_Contact( #TMP_EnTension.QU )
   END_RUNG wire#w1
   RUNG wire#powerrail
      I_Contact( #EnTension )
   END_RUNG wire#w2
   // the same network as SCL:
   #TMP_EnTension(IN := #EnTension AND NOT #TMP_EnTension.QU,   // "FB910_CNT_UHS"
                  R := NOT #EnTension,
                  PV := "V_TMP_EsperaEnTension",
                  BaseUnidades_ms := "CTE_BaseUnidades_1ms");
END_REGION

REGION Network 41: ERROR - Termico de Elevacion
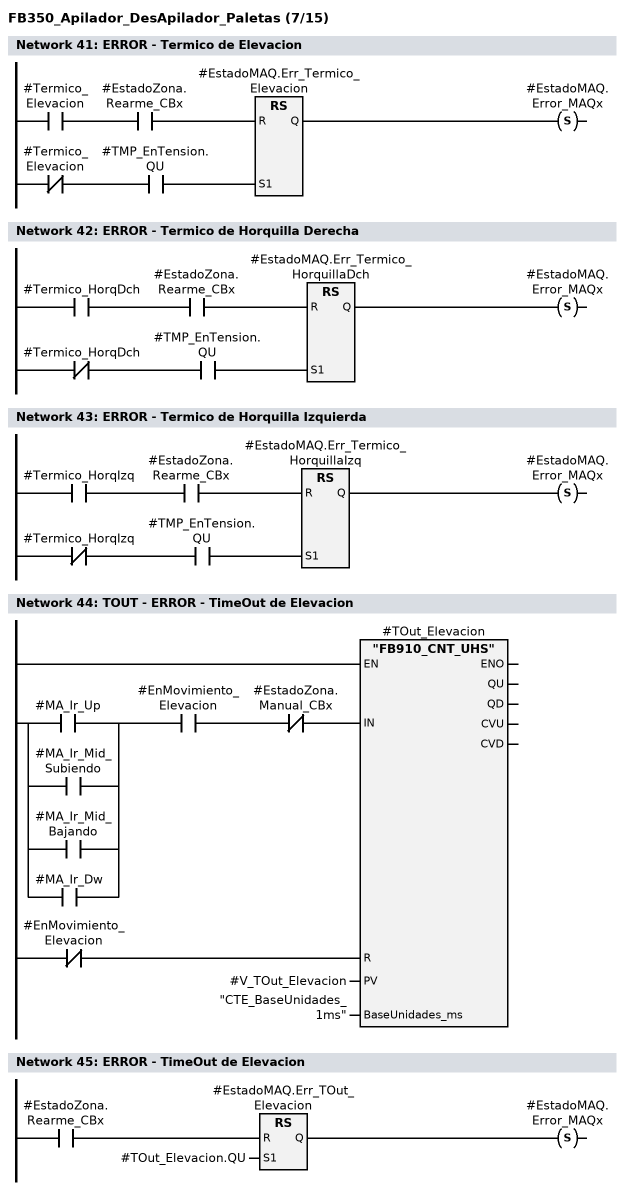
   RUNG wire#powerrail
      Contact( #Termico_Elevacion )
      Contact( #EstadoZona.Rearme_CBx )
      S_RS(operand := #EstadoMAQ.Err_Termico_Elevacion, s1 := wire#w1)
      S_Coil( #EstadoMAQ.Error_MAQx )
   END_RUNG
   RUNG wire#powerrail
      I_Contact( #Termico_Elevacion )
      Contact( #TMP_EnTension.QU )
   END_RUNG wire#w1
   // the same network as SCL:
   IF #Termico_Elevacion AND #EstadoZona.Rearme_CBx THEN
       #EstadoMAQ.Err_Termico_Elevacion := FALSE;   // RS flip-flop
   END_IF;
   IF NOT #Termico_Elevacion AND #TMP_EnTension.QU THEN #EstadoMAQ.Err_Termico_Elevacion := TRUE; END_IF;
   IF #EstadoMAQ.Err_Termico_Elevacion THEN #EstadoMAQ.Error_MAQx := TRUE; END_IF;
END_REGION

REGION Network 42: ERROR - Termico de Horquilla Derecha
   RUNG wire#powerrail
      Contact( #Termico_HorqDch )
      Contact( #EstadoZona.Rearme_CBx )
      S_RS(operand := #EstadoMAQ.Err_Termico_HorquillaDch, s1 := wire#w1)
      S_Coil( #EstadoMAQ.Error_MAQx )
   END_RUNG
   RUNG wire#powerrail
      I_Contact( #Termico_HorqDch )
      Contact( #TMP_EnTension.QU )
   END_RUNG wire#w1
   // the same network as SCL:
   IF #Termico_HorqDch AND #EstadoZona.Rearme_CBx THEN
       #EstadoMAQ.Err_Termico_HorquillaDch := FALSE;   // RS flip-flop
   END_IF;
   IF NOT #Termico_HorqDch AND #TMP_EnTension.QU THEN #EstadoMAQ.Err_Termico_HorquillaDch := TRUE; END_IF;
   IF #EstadoMAQ.Err_Termico_HorquillaDch THEN #EstadoMAQ.Error_MAQx := TRUE; END_IF;
END_REGION

REGION Network 43: ERROR - Termico de Horquilla Izquierda
   RUNG wire#powerrail
      Contact( #Termico_HorqIzq )
      Contact( #EstadoZona.Rearme_CBx )
      S_RS(operand := #EstadoMAQ.Err_Termico_HorquillaIzq, s1 := wire#w1)
      S_Coil( #EstadoMAQ.Error_MAQx )
   END_RUNG
   RUNG wire#powerrail
      I_Contact( #Termico_HorqIzq )
      Contact( #TMP_EnTension.QU )
   END_RUNG wire#w1
   // the same network as SCL:
   IF #Termico_HorqIzq AND #EstadoZona.Rearme_CBx THEN
       #EstadoMAQ.Err_Termico_HorquillaIzq := FALSE;   // RS flip-flop
   END_IF;
   IF NOT #Termico_HorqIzq AND #TMP_EnTension.QU THEN #EstadoMAQ.Err_Termico_HorquillaIzq := TRUE; END_IF;
   IF #EstadoMAQ.Err_Termico_HorquillaIzq THEN #EstadoMAQ.Error_MAQx := TRUE; END_IF;
END_REGION

REGION Network 44: TOUT - ERROR - TimeOut de Elevacion
   RUNG wire#powerrail
      #TOut_Elevacion(IN := wire#w2, R := wire#w3, PV := #V_TOut_Elevacion, BaseUnidades_ms := "CTE_BaseUnidades_1ms", QU =>, QD =>, CVU =>, CVD =>)
   END_RUNG
   RUNG wire#powerrail
      Contact( #MA_Ir_Up )
      wire#w1
      Contact( #EnMovimiento_Elevacion )
      I_Contact( #EstadoZona.Manual_CBx )
   END_RUNG wire#w2
   RUNG wire#powerrail
      Contact( #MA_Ir_Mid_Subiendo )
   END_RUNG wire#w1
   RUNG wire#powerrail
      Contact( #MA_Ir_Mid_Bajando )
   END_RUNG wire#w1
   RUNG wire#powerrail
      Contact( #MA_Ir_Dw )
   END_RUNG wire#w1
   RUNG wire#powerrail
      I_Contact( #EnMovimiento_Elevacion )
   END_RUNG wire#w3
   // the same network as SCL:
   #TOut_Elevacion(IN := (#MA_Ir_Up OR #MA_Ir_Mid_Subiendo OR #MA_Ir_Mid_Bajando OR #MA_Ir_Dw) AND #EnMovimiento_Elevacion AND NOT #EstadoZona.Manual_CBx,   // "FB910_CNT_UHS"
                   R := NOT #EnMovimiento_Elevacion,
                   PV := #V_TOut_Elevacion,
                   BaseUnidades_ms := "CTE_BaseUnidades_1ms");
END_REGION

REGION Network 45: ERROR - TimeOut de Elevacion
   RUNG wire#powerrail
      Contact( #EstadoZona.Rearme_CBx )
      S_RS(operand := #EstadoMAQ.Err_TOut_Elevacion, s1 := #TOut_Elevacion.QU)
      S_Coil( #EstadoMAQ.Error_MAQx )
   END_RUNG
   // the same network as SCL:
   IF #EstadoZona.Rearme_CBx THEN
       #EstadoMAQ.Err_TOut_Elevacion := FALSE;   // RS flip-flop
   END_IF;
   IF #TOut_Elevacion.QU THEN #EstadoMAQ.Err_TOut_Elevacion := TRUE; END_IF;
   IF #EstadoMAQ.Err_TOut_Elevacion THEN #EstadoMAQ.Error_MAQx := TRUE; END_IF;
END_REGION

REGION Network 46: TOUT - ERROR - TimeOut de Horqillado - Abriendo o Cerrando la Horquilla
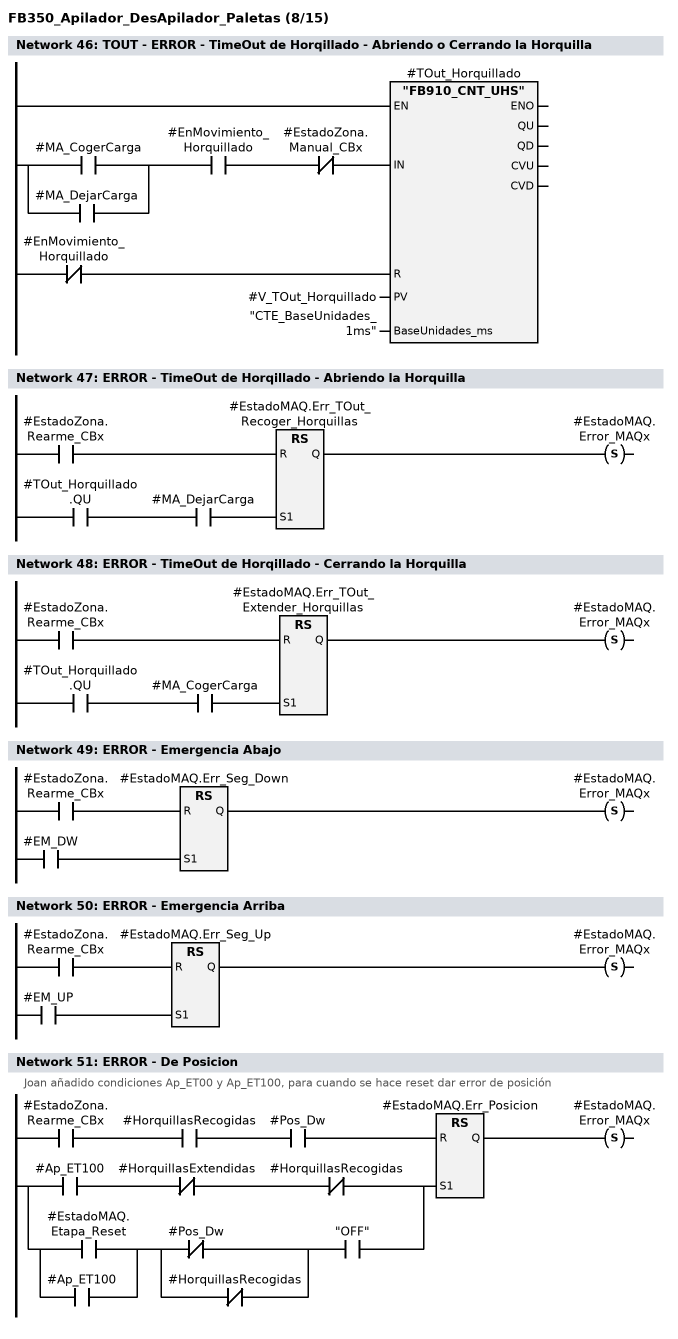
   RUNG wire#powerrail
      #TOut_Horquillado(IN := wire#w2, R := wire#w3, PV := #V_TOut_Horquillado, BaseUnidades_ms := "CTE_BaseUnidades_1ms", QU =>, QD =>, CVU =>, CVD =>)
   END_RUNG
   RUNG wire#powerrail
      Contact( #MA_CogerCarga )
      wire#w1
      Contact( #EnMovimiento_Horquillado )
      I_Contact( #EstadoZona.Manual_CBx )
   END_RUNG wire#w2
   RUNG wire#powerrail
      Contact( #MA_DejarCarga )
   END_RUNG wire#w1
   RUNG wire#powerrail
      I_Contact( #EnMovimiento_Horquillado )
   END_RUNG wire#w3
   // the same network as SCL:
   #TOut_Horquillado(IN := (#MA_CogerCarga OR #MA_DejarCarga) AND #EnMovimiento_Horquillado AND NOT #EstadoZona.Manual_CBx,   // "FB910_CNT_UHS"
                     R := NOT #EnMovimiento_Horquillado,
                     PV := #V_TOut_Horquillado,
                     BaseUnidades_ms := "CTE_BaseUnidades_1ms");
END_REGION

REGION Network 47: ERROR - TimeOut de Horqillado - Abriendo la Horquilla
   RUNG wire#powerrail
      Contact( #EstadoZona.Rearme_CBx )
      S_RS(operand := #EstadoMAQ.Err_TOut_Recoger_Horquillas, s1 := wire#w1)
      S_Coil( #EstadoMAQ.Error_MAQx )
   END_RUNG
   RUNG wire#powerrail
      Contact( #TOut_Horquillado.QU )
      Contact( #MA_DejarCarga )
   END_RUNG wire#w1
   // the same network as SCL:
   IF #EstadoZona.Rearme_CBx THEN
       #EstadoMAQ.Err_TOut_Recoger_Horquillas := FALSE;   // RS flip-flop
   END_IF;
   IF #TOut_Horquillado.QU AND #MA_DejarCarga THEN #EstadoMAQ.Err_TOut_Recoger_Horquillas := TRUE; END_IF;
   IF #EstadoMAQ.Err_TOut_Recoger_Horquillas THEN #EstadoMAQ.Error_MAQx := TRUE; END_IF;
END_REGION

REGION Network 48: ERROR - TimeOut de Horqillado - Cerrando la Horquilla
   RUNG wire#powerrail
      Contact( #EstadoZona.Rearme_CBx )
      S_RS(operand := #EstadoMAQ.Err_TOut_Extender_Horquillas, s1 := wire#w1)
      S_Coil( #EstadoMAQ.Error_MAQx )
   END_RUNG
   RUNG wire#powerrail
      Contact( #TOut_Horquillado.QU )
      Contact( #MA_CogerCarga )
   END_RUNG wire#w1
   // the same network as SCL:
   IF #EstadoZona.Rearme_CBx THEN
       #EstadoMAQ.Err_TOut_Extender_Horquillas := FALSE;   // RS flip-flop
   END_IF;
   IF #TOut_Horquillado.QU AND #MA_CogerCarga THEN #EstadoMAQ.Err_TOut_Extender_Horquillas := TRUE; END_IF;
   IF #EstadoMAQ.Err_TOut_Extender_Horquillas THEN #EstadoMAQ.Error_MAQx := TRUE; END_IF;
END_REGION

REGION Network 49: ERROR - Emergencia Abajo
   RUNG wire#powerrail
      Contact( #EstadoZona.Rearme_CBx )
      S_RS(operand := #EstadoMAQ.Err_Seg_Down, s1 := wire#w1)
      S_Coil( #EstadoMAQ.Error_MAQx )
   END_RUNG
   RUNG wire#powerrail
      Contact( #EM_DW )
   END_RUNG wire#w1
   // the same network as SCL:
   IF #EstadoZona.Rearme_CBx THEN
       #EstadoMAQ.Err_Seg_Down := FALSE;   // RS flip-flop
   END_IF;
   IF #EM_DW THEN #EstadoMAQ.Err_Seg_Down := TRUE; END_IF;
   IF #EstadoMAQ.Err_Seg_Down THEN #EstadoMAQ.Error_MAQx := TRUE; END_IF;
END_REGION

REGION Network 50: ERROR - Emergencia Arriba
   RUNG wire#powerrail
      Contact( #EstadoZona.Rearme_CBx )
      S_RS(operand := #EstadoMAQ.Err_Seg_Up, s1 := wire#w1)
      S_Coil( #EstadoMAQ.Error_MAQx )
   END_RUNG
   RUNG wire#powerrail
      Contact( #EM_UP )
   END_RUNG wire#w1
   // the same network as SCL:
   IF #EstadoZona.Rearme_CBx THEN
       #EstadoMAQ.Err_Seg_Up := FALSE;   // RS flip-flop
   END_IF;
   IF #EM_UP THEN #EstadoMAQ.Err_Seg_Up := TRUE; END_IF;
   IF #EstadoMAQ.Err_Seg_Up THEN #EstadoMAQ.Error_MAQx := TRUE; END_IF;
END_REGION

REGION Network 51: ERROR - De Posicion
   // Joan añadido condiciones Ap_ET00 y Ap_ET100, para cuando se hace reset dar error de posición
   RUNG wire#powerrail
      Contact( #EstadoZona.Rearme_CBx )
      Contact( #HorquillasRecogidas )
      Contact( #Pos_Dw )
      S_RS(operand := #EstadoMAQ.Err_Posicion, s1 := wire#w3)
      S_Coil( #EstadoMAQ.Error_MAQx )
   END_RUNG
   RUNG wire#powerrail
      Contact( #Ap_ET100 )
      I_Contact( #HorquillasExtendidas )
      I_Contact( #HorquillasRecogidas )
   END_RUNG wire#w3
   RUNG wire#powerrail
      Contact( #EstadoMAQ.Etapa_Reset )
      wire#w1
      I_Contact( #Pos_Dw )
      wire#w2
      Contact( "OFF" )
   END_RUNG wire#w3
   RUNG wire#powerrail
      Contact( #Ap_ET100 )
   END_RUNG wire#w1
   RUNG wire#w1
      I_Contact( #HorquillasRecogidas )
   END_RUNG wire#w2
   // the same network as SCL:
   IF #EstadoZona.Rearme_CBx AND #HorquillasRecogidas AND #Pos_Dw THEN
       #EstadoMAQ.Err_Posicion := FALSE;   // RS flip-flop
   END_IF;
   IF (#Ap_ET100 AND NOT #HorquillasExtendidas AND NOT #HorquillasRecogidas) OR ((#EstadoMAQ.Etapa_Reset OR #Ap_ET100) AND (NOT #Pos_Dw OR NOT #HorquillasRecogidas) AND "OFF") THEN
       #EstadoMAQ.Err_Posicion := TRUE;
   END_IF;
   IF #EstadoMAQ.Err_Posicion THEN #EstadoMAQ.Error_MAQx := TRUE; END_IF;
END_REGION

REGION Network 52: TEMPORIZADOR - ESTABILIDAD para Fin de los Movimientos
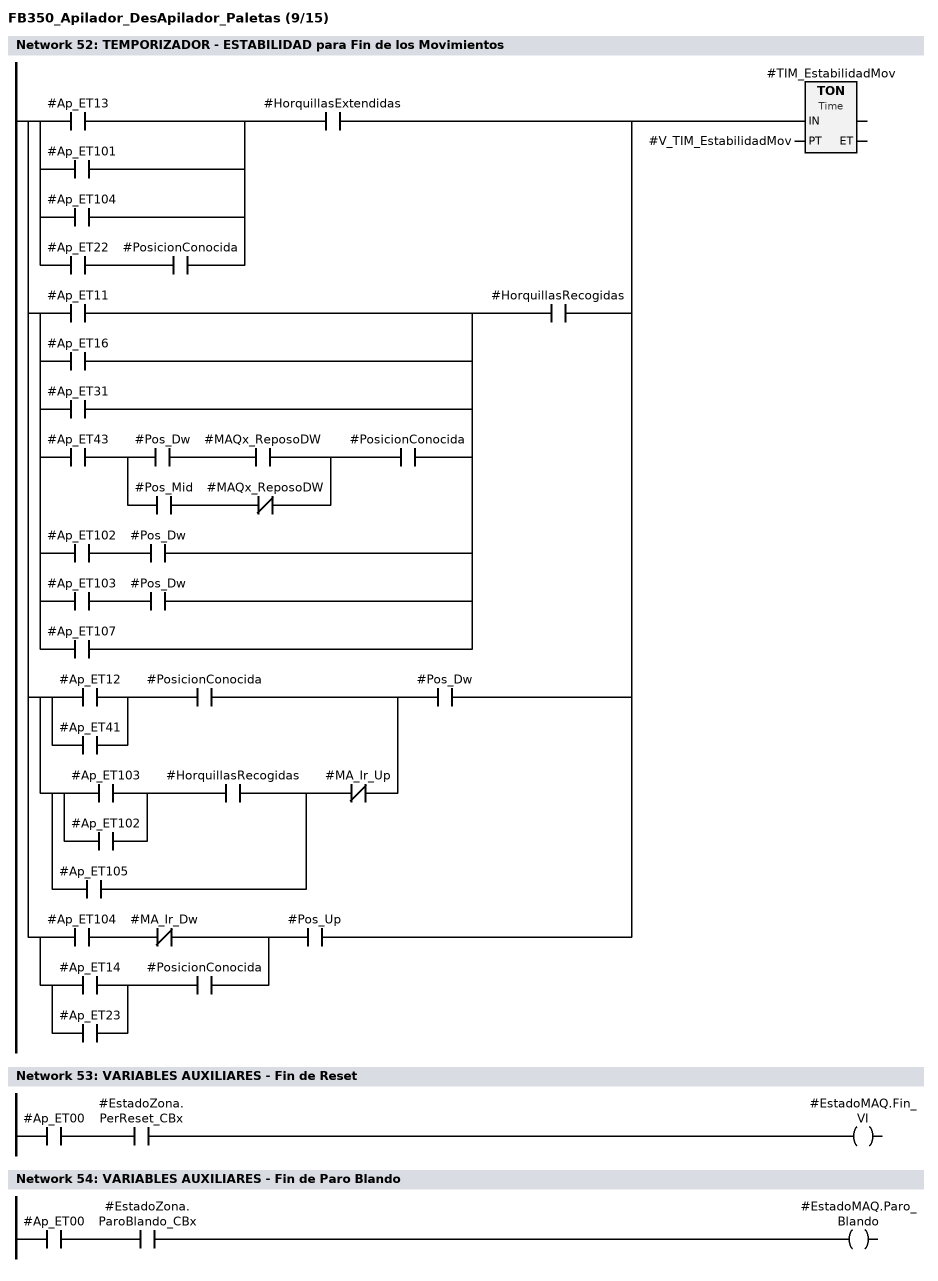
   RUNG wire#powerrail
      Contact( #Ap_ET13 )
      wire#w1
      Contact( #HorquillasExtendidas )
      wire#w2
      { S7_Templates := "time_type := Time" } #TIM_EstabilidadMov.TON(pt := #V_TIM_EstabilidadMov, et =>)
   END_RUNG
   RUNG wire#powerrail
      Contact( #Ap_ET101 )
   END_RUNG wire#w1
   RUNG wire#powerrail
      Contact( #Ap_ET104 )
   END_RUNG wire#w1
   RUNG wire#powerrail
      Contact( #Ap_ET22 )
      Contact( #PosicionConocida )
   END_RUNG wire#w1
   RUNG wire#powerrail
      Contact( #Ap_ET11 )
      wire#w3
      Contact( #HorquillasRecogidas )
   END_RUNG wire#w2
   RUNG wire#powerrail
      Contact( #Ap_ET16 )
   END_RUNG wire#w3
   RUNG wire#powerrail
      Contact( #Ap_ET31 )
   END_RUNG wire#w3
   RUNG wire#powerrail
      Contact( #Ap_ET43 )
      wire#w4
      Contact( #Pos_Dw )
      Contact( #MAQx_ReposoDW )
      wire#w5
      Contact( #PosicionConocida )
   END_RUNG wire#w3
   RUNG wire#w4
      Contact( #Pos_Mid )
      I_Contact( #MAQx_ReposoDW )
   END_RUNG wire#w5
   RUNG wire#powerrail
      Contact( #Ap_ET102 )
      Contact( #Pos_Dw )
   END_RUNG wire#w3
   RUNG wire#powerrail
      Contact( #Ap_ET103 )
      Contact( #Pos_Dw )
   END_RUNG wire#w3
   RUNG wire#powerrail
      Contact( #Ap_ET107 )
   END_RUNG wire#w3
   RUNG wire#powerrail
      Contact( #Ap_ET12 )
      wire#w6
      Contact( #PosicionConocida )
      wire#w7
      Contact( #Pos_Dw )
   END_RUNG wire#w2
   RUNG wire#powerrail
      Contact( #Ap_ET41 )
   END_RUNG wire#w6
   RUNG wire#powerrail
      Contact( #Ap_ET103 )
      wire#w8
      Contact( #HorquillasRecogidas )
      wire#w9
      I_Contact( #MA_Ir_Up )
   END_RUNG wire#w7
   RUNG wire#powerrail
      Contact( #Ap_ET102 )
   END_RUNG wire#w8
   RUNG wire#powerrail
      Contact( #Ap_ET105 )
   END_RUNG wire#w9
   RUNG wire#powerrail
      Contact( #Ap_ET104 )
      I_Contact( #MA_Ir_Dw )
      wire#w10
      Contact( #Pos_Up )
   END_RUNG wire#w2
   RUNG wire#powerrail
      Contact( #Ap_ET14 )
      wire#w11
      Contact( #PosicionConocida )
   END_RUNG wire#w10
   RUNG wire#powerrail
      Contact( #Ap_ET23 )
   END_RUNG wire#w11
   // the same network as SCL:
   #TIM_EstabilidadMov(IN := ((#Ap_ET13 OR #Ap_ET101 OR #Ap_ET104 OR (#Ap_ET22 AND #PosicionConocida)) AND #HorquillasExtendidas) OR ((#Ap_ET11 OR #Ap_ET16 OR #Ap_ET31 OR (#Ap_ET43 AND ((#Pos_Dw AND #MAQx_ReposoDW) OR (#Pos_Mid AND NOT #MAQx_ReposoDW)) AND #PosicionConocida) OR (#Ap_ET102 AND #Pos_Dw) OR (#Ap_ET103 AND #Pos_Dw) OR #Ap_ET107) AND #HorquillasRecogidas) OR ((((#Ap_ET12 OR #Ap_ET41) AND #PosicionConocida) OR ((((#Ap_ET103 OR #Ap_ET102) AND #HorquillasRecogidas) OR #Ap_ET105) AND NOT #MA_Ir_Up)) AND #Pos_Dw) OR (((#Ap_ET104 AND NOT #MA_Ir_Dw) OR ((#Ap_ET14 OR #Ap_ET23) AND #PosicionConocida)) AND #Pos_Up),   // TON
                       PT := #V_TIM_EstabilidadMov);
END_REGION

REGION Network 53: VARIABLES AUXILIARES - Fin de Reset
   RUNG wire#powerrail
      Contact( #Ap_ET00 )
      Contact( #EstadoZona.PerReset_CBx )
      Coil( #EstadoMAQ.Fin_VI )
   END_RUNG
   // the same network as SCL:
   #EstadoMAQ.Fin_VI := #Ap_ET00 AND #EstadoZona.PerReset_CBx;
END_REGION

REGION Network 54: VARIABLES AUXILIARES - Fin de Paro Blando
   RUNG wire#powerrail
      Contact( #Ap_ET00 )
      Contact( #EstadoZona.ParoBlando_CBx )
      Coil( #EstadoMAQ.Paro_Blando )
   END_RUNG
   // the same network as SCL:
   #EstadoMAQ.Paro_Blando := #Ap_ET00 AND #EstadoZona.ParoBlando_CBx;
END_REGION

REGION Network 55: VARIABLES AUXILIARES - Posicion Conocida
   // MODIFICACION DANI: SI MUEVO EN MANUAL NO PIERDE LA POSCION
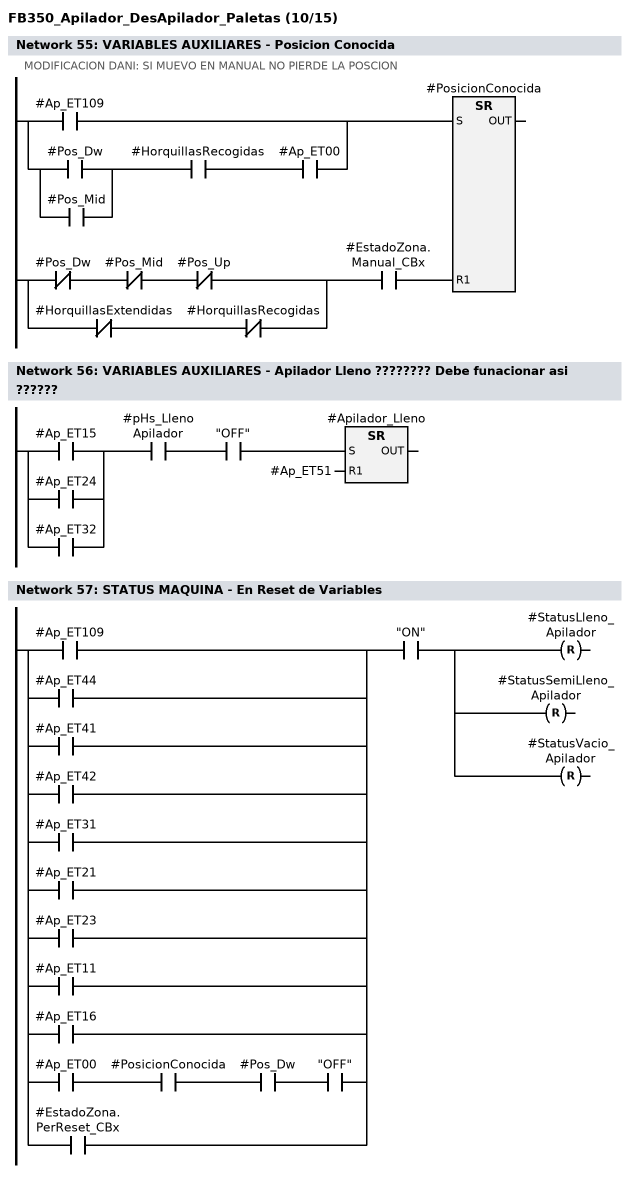
   RUNG wire#powerrail
      Contact( #Ap_ET109 )
      wire#w1
      S_SR(operand := #PosicionConocida, r1 := wire#w4)
   END_RUNG
   RUNG wire#powerrail
      Contact( #Pos_Dw )
      wire#w2
      Contact( #HorquillasRecogidas )
      Contact( #Ap_ET00 )
   END_RUNG wire#w1
   RUNG wire#powerrail
      Contact( #Pos_Mid )
   END_RUNG wire#w2
   RUNG wire#powerrail
      I_Contact( #Pos_Dw )
      I_Contact( #Pos_Mid )
      I_Contact( #Pos_Up )
      wire#w3
      Contact( #EstadoZona.Manual_CBx )
   END_RUNG wire#w4
   RUNG wire#powerrail
      I_Contact( #HorquillasExtendidas )
      I_Contact( #HorquillasRecogidas )
   END_RUNG wire#w3
   // the same network as SCL:
   IF #Ap_ET109 OR ((#Pos_Dw OR #Pos_Mid) AND #HorquillasRecogidas AND #Ap_ET00) THEN
       #PosicionConocida := TRUE;   // SR flip-flop
   END_IF;
   IF ((NOT #Pos_Dw AND NOT #Pos_Mid AND NOT #Pos_Up) OR (NOT #HorquillasExtendidas AND NOT #HorquillasRecogidas)) AND #EstadoZona.Manual_CBx THEN
       #PosicionConocida := FALSE;
   END_IF;
END_REGION

REGION Network 56: VARIABLES AUXILIARES - Apilador Lleno ???????? Debe funacionar asi ??????
   RUNG wire#powerrail
      Contact( #Ap_ET15 )
      wire#w1
      Contact( #pHs_LlenoApilador )
      Contact( "OFF" )
      S_SR(operand := #Apilador_Lleno, r1 := #Ap_ET51)
   END_RUNG
   RUNG wire#powerrail
      Contact( #Ap_ET24 )
   END_RUNG wire#w1
   RUNG wire#powerrail
      Contact( #Ap_ET32 )
   END_RUNG wire#w1
   // the same network as SCL:
   IF (#Ap_ET15 OR #Ap_ET24 OR #Ap_ET32) AND #pHs_LlenoApilador AND "OFF" THEN
       #Apilador_Lleno := TRUE;   // SR flip-flop
   END_IF;
   IF #Ap_ET51 THEN #Apilador_Lleno := FALSE; END_IF;
END_REGION

REGION Network 57: STATUS MAQUINA - En Reset de Variables
   RUNG wire#powerrail
      Contact( #Ap_ET109 )
      wire#w1
      Contact( "ON" )
      wire#w2
      R_Coil( #StatusLleno_Apilador )
   END_RUNG
   RUNG wire#powerrail
      Contact( #Ap_ET44 )
   END_RUNG wire#w1
   RUNG wire#powerrail
      Contact( #Ap_ET41 )
   END_RUNG wire#w1
   RUNG wire#powerrail
      Contact( #Ap_ET42 )
   END_RUNG wire#w1
   RUNG wire#powerrail
      Contact( #Ap_ET31 )
   END_RUNG wire#w1
   RUNG wire#powerrail
      Contact( #Ap_ET21 )
   END_RUNG wire#w1
   RUNG wire#powerrail
      Contact( #Ap_ET23 )
   END_RUNG wire#w1
   RUNG wire#powerrail
      Contact( #Ap_ET11 )
   END_RUNG wire#w1
   RUNG wire#powerrail
      Contact( #Ap_ET16 )
   END_RUNG wire#w1
   RUNG wire#powerrail
      Contact( #Ap_ET00 )
      Contact( #PosicionConocida )
      Contact( #Pos_Dw )
      Contact( "OFF" )
   END_RUNG wire#w1
   RUNG wire#powerrail
      Contact( #EstadoZona.PerReset_CBx )
   END_RUNG wire#w1
   RUNG wire#w2
      R_Coil( #StatusSemiLleno_Apilador )
   END_RUNG
   RUNG wire#w2
      R_Coil( #StatusVacio_Apilador )
   END_RUNG
   // the same network as SCL:
   IF (#Ap_ET109 OR #Ap_ET44 OR #Ap_ET41 OR #Ap_ET42 OR #Ap_ET31 OR #Ap_ET21 OR #Ap_ET23 OR #Ap_ET11 OR #Ap_ET16 OR (#Ap_ET00 AND #PosicionConocida AND #Pos_Dw AND "OFF") OR #EstadoZona.PerReset_CBx) AND "ON" THEN
       #StatusLleno_Apilador := FALSE;
       #StatusSemiLleno_Apilador := FALSE;
       #StatusVacio_Apilador := FALSE;
   END_IF;
END_REGION

REGION Network 58: STATUS MAQUINA - En set de Variables
   // DANI SI ESTA EN ETAPA 0, POS CONOCIDA Y POS REPOSO ACTUALICE EL ESTATUS
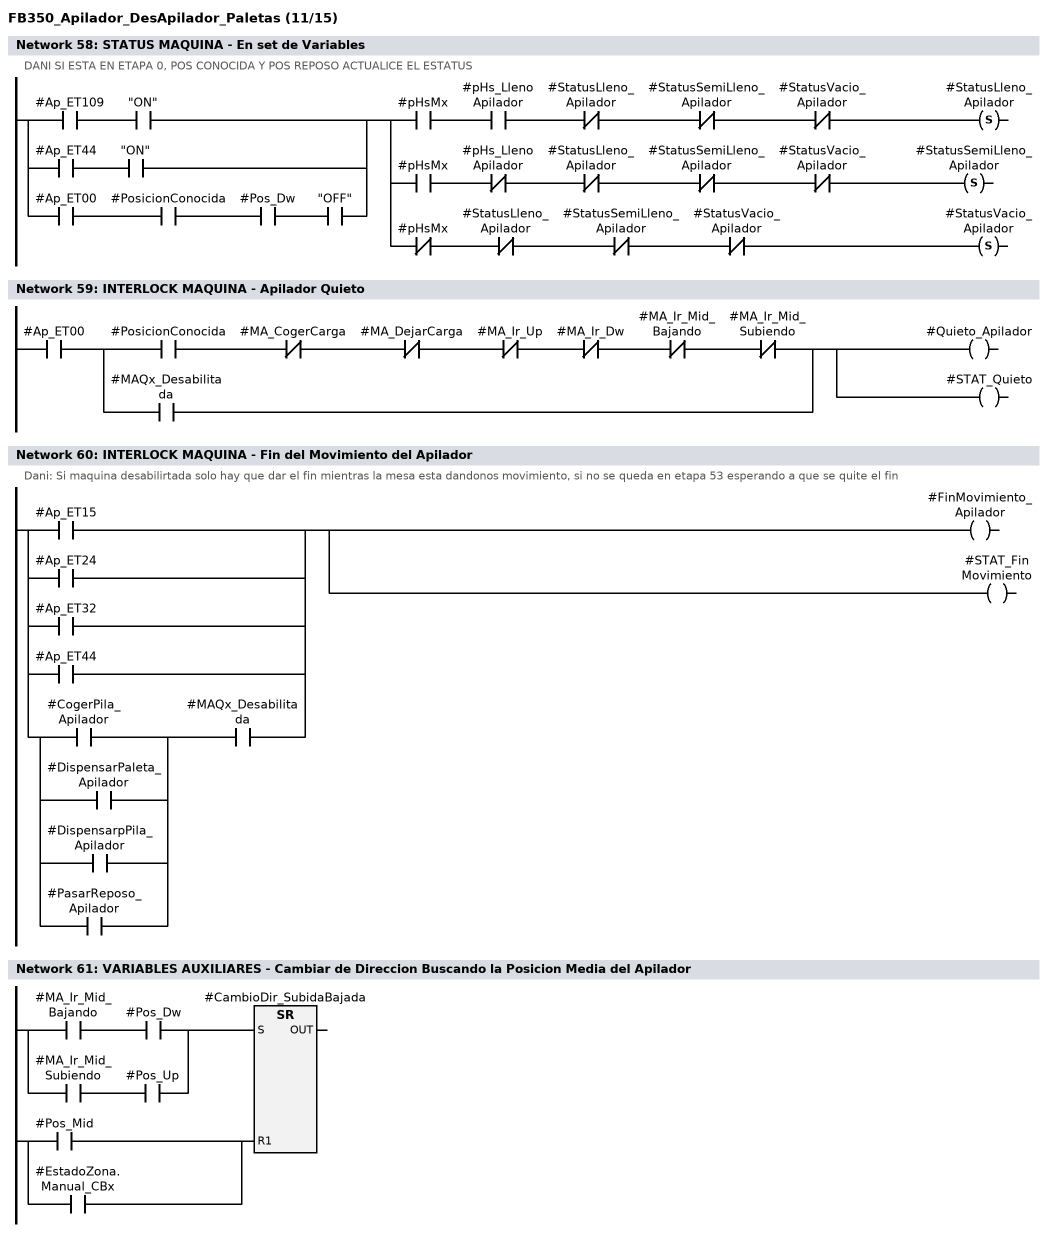
   RUNG wire#powerrail
      Contact( #Ap_ET109 )
      Contact( "ON" )
      wire#w1
      Contact( #pHsMx )
      Contact( #pHs_LlenoApilador )
      I_Contact( #StatusLleno_Apilador )
      I_Contact( #StatusSemiLleno_Apilador )
      I_Contact( #StatusVacio_Apilador )
      S_Coil( #StatusLleno_Apilador )
   END_RUNG
   RUNG wire#powerrail
      Contact( #Ap_ET44 )
      Contact( "ON" )
   END_RUNG wire#w1
   RUNG wire#powerrail
      Contact( #Ap_ET00 )
      Contact( #PosicionConocida )
      Contact( #Pos_Dw )
      Contact( "OFF" )
   END_RUNG wire#w1
   RUNG wire#w1
      Contact( #pHsMx )
      I_Contact( #pHs_LlenoApilador )
      I_Contact( #StatusLleno_Apilador )
      I_Contact( #StatusSemiLleno_Apilador )
      I_Contact( #StatusVacio_Apilador )
      S_Coil( #StatusSemiLleno_Apilador )
   END_RUNG
   RUNG wire#w1
      I_Contact( #pHsMx )
      I_Contact( #StatusLleno_Apilador )
      I_Contact( #StatusSemiLleno_Apilador )
      I_Contact( #StatusVacio_Apilador )
      S_Coil( #StatusVacio_Apilador )
   END_RUNG
   // the same network as SCL:
   #_w1 := (#Ap_ET109 AND "ON") OR (#Ap_ET44 AND "ON") OR (#Ap_ET00 AND #PosicionConocida AND #Pos_Dw AND "OFF");
   IF #_w1 AND #pHsMx AND #pHs_LlenoApilador AND NOT #StatusLleno_Apilador AND NOT #StatusSemiLleno_Apilador AND NOT #StatusVacio_Apilador THEN
       #StatusLleno_Apilador := TRUE;
   END_IF;
   IF #_w1 AND #pHsMx AND NOT #pHs_LlenoApilador AND NOT #StatusLleno_Apilador AND NOT #StatusSemiLleno_Apilador AND NOT #StatusVacio_Apilador THEN
       #StatusSemiLleno_Apilador := TRUE;
   END_IF;
   IF #_w1 AND NOT #pHsMx AND NOT #StatusLleno_Apilador AND NOT #StatusSemiLleno_Apilador AND NOT #StatusVacio_Apilador THEN
       #StatusVacio_Apilador := TRUE;
   END_IF;
END_REGION

REGION Network 59: INTERLOCK MAQUINA - Apilador Quieto
   RUNG wire#powerrail
      Contact( #Ap_ET00 )
      wire#w1
      Contact( #PosicionConocida )
      I_Contact( #MA_CogerCarga )
      I_Contact( #MA_DejarCarga )
      I_Contact( #MA_Ir_Up )
      I_Contact( #MA_Ir_Dw )
      I_Contact( #MA_Ir_Mid_Bajando )
      I_Contact( #MA_Ir_Mid_Subiendo )
      wire#w2
      Coil( #Quieto_Apilador )
   END_RUNG
   RUNG wire#w1
      Contact( #MAQx_Desabilitada )
   END_RUNG wire#w2
   RUNG wire#w2
      Coil( #STAT_Quieto )
   END_RUNG
   // the same network as SCL:
   #Quieto_Apilador := #Ap_ET00 AND ((#PosicionConocida AND NOT #MA_CogerCarga AND NOT #MA_DejarCarga AND NOT #MA_Ir_Up AND NOT #MA_Ir_Dw AND NOT #MA_Ir_Mid_Bajando AND NOT #MA_Ir_Mid_Subiendo) OR #MAQx_Desabilitada);
   #STAT_Quieto := #Quieto_Apilador;
END_REGION

REGION Network 60: INTERLOCK MAQUINA - Fin del Movimiento del Apilador
   // Dani: Si maquina desabilirtada solo hay que dar el fin mientras la mesa esta dandonos movimiento, si no se queda en etapa 53 esperando a que se quite el fin
   RUNG wire#powerrail
      Contact( #Ap_ET15 )
      wire#w1
      Coil( #FinMovimiento_Apilador )
   END_RUNG
   RUNG wire#powerrail
      Contact( #Ap_ET24 )
   END_RUNG wire#w1
   RUNG wire#powerrail
      Contact( #Ap_ET32 )
   END_RUNG wire#w1
   RUNG wire#powerrail
      Contact( #Ap_ET44 )
   END_RUNG wire#w1
   RUNG wire#powerrail
      Contact( #CogerPila_Apilador )
      wire#w2
      Contact( #MAQx_Desabilitada )
   END_RUNG wire#w1
   RUNG wire#powerrail
      Contact( #DispensarPaleta_Apilador )
   END_RUNG wire#w2
   RUNG wire#powerrail
      Contact( #DispensarpPila_Apilador )
   END_RUNG wire#w2
   RUNG wire#powerrail
      Contact( #PasarReposo_Apilador )
   END_RUNG wire#w2
   RUNG wire#w1
      Coil( #STAT_FinMovimiento )
   END_RUNG
   // the same network as SCL:
   #FinMovimiento_Apilador := #Ap_ET15 OR #Ap_ET24 OR #Ap_ET32 OR #Ap_ET44 OR ((#CogerPila_Apilador OR #DispensarPaleta_Apilador OR #DispensarpPila_Apilador OR #PasarReposo_Apilador) AND #MAQx_Desabilitada);
   #STAT_FinMovimiento := #FinMovimiento_Apilador;
END_REGION

REGION Network 61: VARIABLES AUXILIARES - Cambiar de Direccion Buscando la Posicion Media del Apilador
   RUNG wire#powerrail
      Contact( #MA_Ir_Mid_Bajando )
      Contact( #Pos_Dw )
      wire#w1
      S_SR(operand := #CambioDir_SubidaBajada, r1 := wire#w2)
   END_RUNG
   RUNG wire#powerrail
      Contact( #MA_Ir_Mid_Subiendo )
      Contact( #Pos_Up )
   END_RUNG wire#w1
   RUNG wire#powerrail
      Contact( #Pos_Mid )
   END_RUNG wire#w2
   RUNG wire#powerrail
      Contact( #EstadoZona.Manual_CBx )
   END_RUNG wire#w2
   // the same network as SCL:
   IF (#MA_Ir_Mid_Bajando AND #Pos_Dw) OR (#MA_Ir_Mid_Subiendo AND #Pos_Up) THEN
       #CambioDir_SubidaBajada := TRUE;   // SR flip-flop
   END_IF;
   IF #Pos_Mid OR #EstadoZona.Manual_CBx THEN #CambioDir_SubidaBajada := FALSE; END_IF;
END_REGION

REGION Network 62: SALIDAS EXTERIORES - Hoquilla - Coger Carga / Extender 4 Horquillas
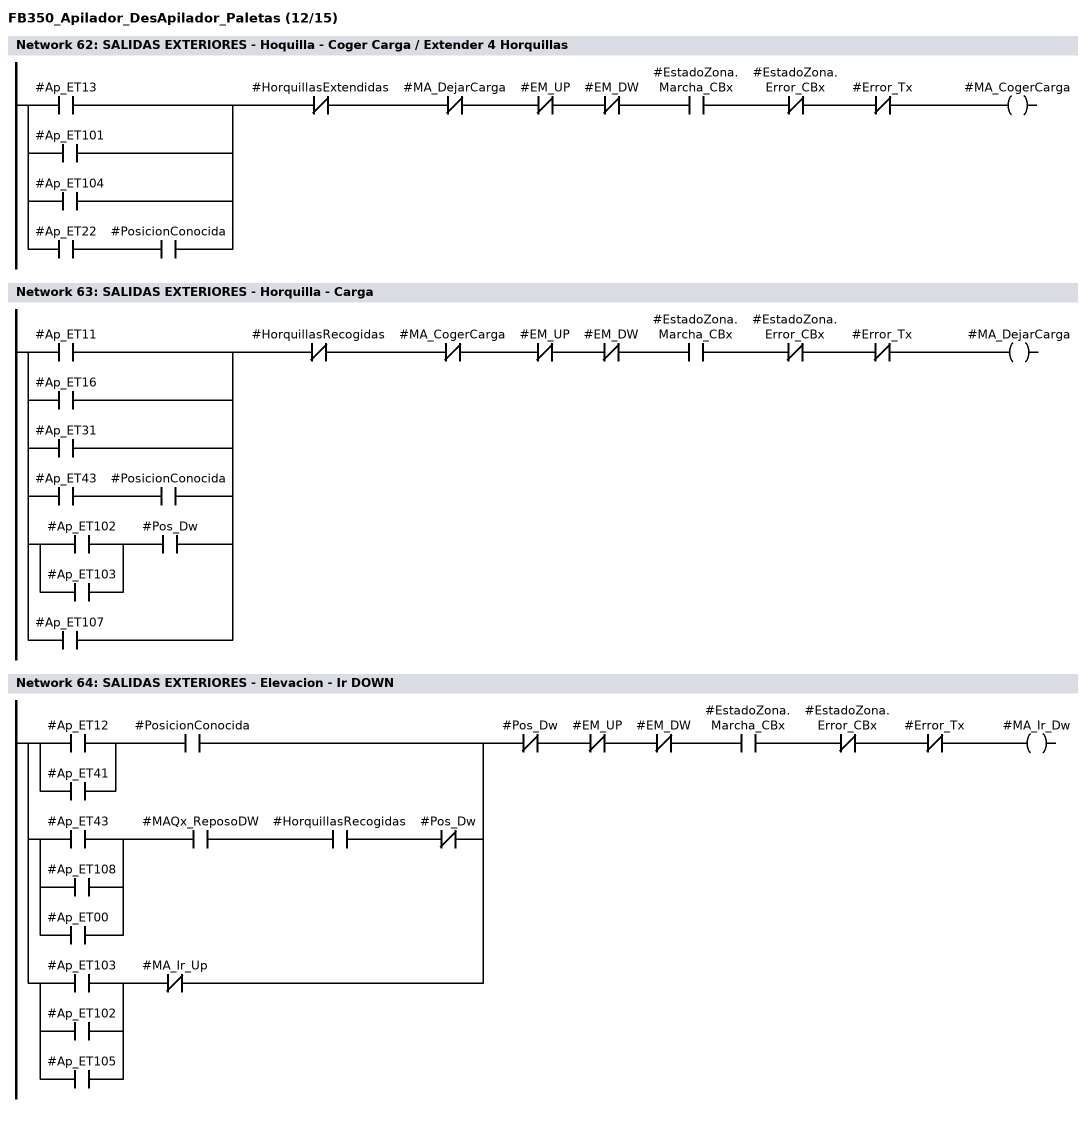
   RUNG wire#powerrail
      Contact( #Ap_ET13 )
      wire#w1
      I_Contact( #HorquillasExtendidas )
      I_Contact( #MA_DejarCarga )
      I_Contact( #EM_UP )
      I_Contact( #EM_DW )
      Contact( #EstadoZona.Marcha_CBx )
      I_Contact( #EstadoZona.Error_CBx )
      I_Contact( #Error_Tx )
      Coil( #MA_CogerCarga )
   END_RUNG
   RUNG wire#powerrail
      Contact( #Ap_ET101 )
   END_RUNG wire#w1
   RUNG wire#powerrail
      Contact( #Ap_ET104 )
   END_RUNG wire#w1
   RUNG wire#powerrail
      Contact( #Ap_ET22 )
      Contact( #PosicionConocida )
   END_RUNG wire#w1
   // the same network as SCL:
   #MA_CogerCarga := (#Ap_ET13 OR #Ap_ET101 OR #Ap_ET104 OR (#Ap_ET22 AND #PosicionConocida)) AND NOT #HorquillasExtendidas AND NOT #MA_DejarCarga AND NOT #EM_UP AND NOT #EM_DW AND #EstadoZona.Marcha_CBx AND NOT #EstadoZona.Error_CBx AND NOT #Error_Tx;
END_REGION

REGION Network 63: SALIDAS EXTERIORES - Horquilla - Carga
   RUNG wire#powerrail
      Contact( #Ap_ET11 )
      wire#w1
      I_Contact( #HorquillasRecogidas )
      I_Contact( #MA_CogerCarga )
      I_Contact( #EM_UP )
      I_Contact( #EM_DW )
      Contact( #EstadoZona.Marcha_CBx )
      I_Contact( #EstadoZona.Error_CBx )
      I_Contact( #Error_Tx )
      Coil( #MA_DejarCarga )
   END_RUNG
   RUNG wire#powerrail
      Contact( #Ap_ET16 )
   END_RUNG wire#w1
   RUNG wire#powerrail
      Contact( #Ap_ET31 )
   END_RUNG wire#w1
   RUNG wire#powerrail
      Contact( #Ap_ET43 )
      Contact( #PosicionConocida )
   END_RUNG wire#w1
   RUNG wire#powerrail
      Contact( #Ap_ET102 )
      wire#w2
      Contact( #Pos_Dw )
   END_RUNG wire#w1
   RUNG wire#powerrail
      Contact( #Ap_ET103 )
   END_RUNG wire#w2
   RUNG wire#powerrail
      Contact( #Ap_ET107 )
   END_RUNG wire#w1
   // the same network as SCL:
   #MA_DejarCarga := (#Ap_ET11 OR #Ap_ET16 OR #Ap_ET31 OR (#Ap_ET43 AND #PosicionConocida) OR ((#Ap_ET102 OR #Ap_ET103) AND #Pos_Dw) OR #Ap_ET107) AND NOT #HorquillasRecogidas AND NOT #MA_CogerCarga AND NOT #EM_UP AND NOT #EM_DW AND #EstadoZona.Marcha_CBx AND NOT #EstadoZona.Error_CBx AND NOT #Error_Tx;
END_REGION

REGION Network 64: SALIDAS EXTERIORES - Elevacion - Ir DOWN
   RUNG wire#powerrail
      Contact( #Ap_ET12 )
      wire#w1
      Contact( #PosicionConocida )
      wire#w2
      I_Contact( #Pos_Dw )
      I_Contact( #EM_UP )
      I_Contact( #EM_DW )
      Contact( #EstadoZona.Marcha_CBx )
      I_Contact( #EstadoZona.Error_CBx )
      I_Contact( #Error_Tx )
      Coil( #MA_Ir_Dw )
   END_RUNG
   RUNG wire#powerrail
      Contact( #Ap_ET41 )
   END_RUNG wire#w1
   RUNG wire#powerrail
      Contact( #Ap_ET43 )
      wire#w3
      Contact( #MAQx_ReposoDW )
      Contact( #HorquillasRecogidas )
      I_Contact( #Pos_Dw )
   END_RUNG wire#w2
   RUNG wire#powerrail
      Contact( #Ap_ET108 )
   END_RUNG wire#w3
   RUNG wire#powerrail
      Contact( #Ap_ET00 )
   END_RUNG wire#w3
   RUNG wire#powerrail
      Contact( #Ap_ET103 )
      wire#w4
      I_Contact( #MA_Ir_Up )
   END_RUNG wire#w2
   RUNG wire#powerrail
      Contact( #Ap_ET102 )
   END_RUNG wire#w4
   RUNG wire#powerrail
      Contact( #Ap_ET105 )
   END_RUNG wire#w4
   // the same network as SCL:
   #MA_Ir_Dw := (((#Ap_ET12 OR #Ap_ET41) AND #PosicionConocida) OR ((#Ap_ET43 OR #Ap_ET108 OR #Ap_ET00) AND #MAQx_ReposoDW AND #HorquillasRecogidas AND NOT #Pos_Dw) OR ((#Ap_ET103 OR #Ap_ET102 OR #Ap_ET105) AND NOT #MA_Ir_Up)) AND NOT #Pos_Dw AND NOT #EM_UP AND NOT #EM_DW AND #EstadoZona.Marcha_CBx AND NOT #EstadoZona.Error_CBx AND NOT #Error_Tx;
END_REGION

REGION Network 65: SALIDAS EXTERIORES - Elevacion - Ir MID Bajando
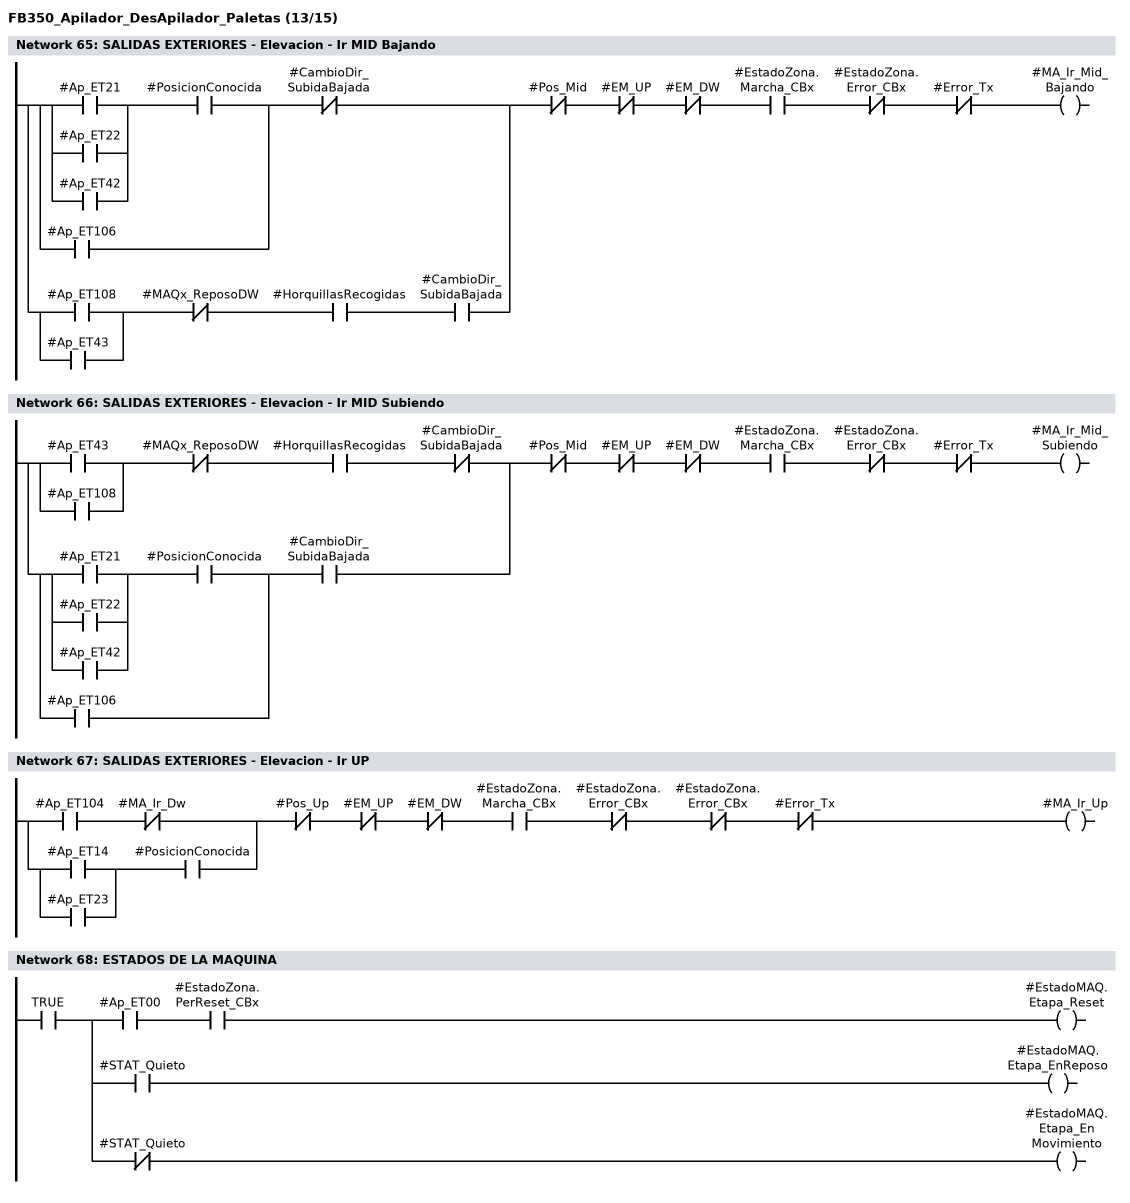
   RUNG wire#powerrail
      Contact( #Ap_ET21 )
      wire#w1
      Contact( #PosicionConocida )
      wire#w2
      I_Contact( #CambioDir_SubidaBajada )
      wire#w3
      I_Contact( #Pos_Mid )
      I_Contact( #EM_UP )
      I_Contact( #EM_DW )
      Contact( #EstadoZona.Marcha_CBx )
      I_Contact( #EstadoZona.Error_CBx )
      I_Contact( #Error_Tx )
      Coil( #MA_Ir_Mid_Bajando )
   END_RUNG
   RUNG wire#powerrail
      Contact( #Ap_ET22 )
   END_RUNG wire#w1
   RUNG wire#powerrail
      Contact( #Ap_ET42 )
   END_RUNG wire#w1
   RUNG wire#powerrail
      Contact( #Ap_ET106 )
   END_RUNG wire#w2
   RUNG wire#powerrail
      Contact( #Ap_ET108 )
      wire#w4
      I_Contact( #MAQx_ReposoDW )
      Contact( #HorquillasRecogidas )
      Contact( #CambioDir_SubidaBajada )
   END_RUNG wire#w3
   RUNG wire#powerrail
      Contact( #Ap_ET43 )
   END_RUNG wire#w4
   // the same network as SCL:
   #MA_Ir_Mid_Bajando := (((((#Ap_ET21 OR #Ap_ET22 OR #Ap_ET42) AND #PosicionConocida) OR #Ap_ET106) AND NOT #CambioDir_SubidaBajada) OR ((#Ap_ET108 OR #Ap_ET43) AND NOT #MAQx_ReposoDW AND #HorquillasRecogidas AND #CambioDir_SubidaBajada)) AND NOT #Pos_Mid AND NOT #EM_UP AND NOT #EM_DW AND #EstadoZona.Marcha_CBx AND NOT #EstadoZona.Error_CBx AND NOT #Error_Tx;
END_REGION

REGION Network 66: SALIDAS EXTERIORES - Elevacion - Ir MID Subiendo
   RUNG wire#powerrail
      Contact( #Ap_ET43 )
      wire#w1
      I_Contact( #MAQx_ReposoDW )
      Contact( #HorquillasRecogidas )
      I_Contact( #CambioDir_SubidaBajada )
      wire#w2
      I_Contact( #Pos_Mid )
      I_Contact( #EM_UP )
      I_Contact( #EM_DW )
      Contact( #EstadoZona.Marcha_CBx )
      I_Contact( #EstadoZona.Error_CBx )
      I_Contact( #Error_Tx )
      Coil( #MA_Ir_Mid_Subiendo )
   END_RUNG
   RUNG wire#powerrail
      Contact( #Ap_ET108 )
   END_RUNG wire#w1
   RUNG wire#powerrail
      Contact( #Ap_ET21 )
      wire#w3
      Contact( #PosicionConocida )
      wire#w4
      Contact( #CambioDir_SubidaBajada )
   END_RUNG wire#w2
   RUNG wire#powerrail
      Contact( #Ap_ET22 )
   END_RUNG wire#w3
   RUNG wire#powerrail
      Contact( #Ap_ET42 )
   END_RUNG wire#w3
   RUNG wire#powerrail
      Contact( #Ap_ET106 )
   END_RUNG wire#w4
   // the same network as SCL:
   #MA_Ir_Mid_Subiendo := (((#Ap_ET43 OR #Ap_ET108) AND NOT #MAQx_ReposoDW AND #HorquillasRecogidas AND NOT #CambioDir_SubidaBajada) OR ((((#Ap_ET21 OR #Ap_ET22 OR #Ap_ET42) AND #PosicionConocida) OR #Ap_ET106) AND #CambioDir_SubidaBajada)) AND NOT #Pos_Mid AND NOT #EM_UP AND NOT #EM_DW AND #EstadoZona.Marcha_CBx AND NOT #EstadoZona.Error_CBx AND NOT #Error_Tx;
END_REGION

REGION Network 67: SALIDAS EXTERIORES - Elevacion - Ir UP
   RUNG wire#powerrail
      Contact( #Ap_ET104 )
      I_Contact( #MA_Ir_Dw )
      wire#w1
      I_Contact( #Pos_Up )
      I_Contact( #EM_UP )
      I_Contact( #EM_DW )
      Contact( #EstadoZona.Marcha_CBx )
      I_Contact( #EstadoZona.Error_CBx )
      I_Contact( #EstadoZona.Error_CBx )
      I_Contact( #Error_Tx )
      Coil( #MA_Ir_Up )
   END_RUNG
   RUNG wire#powerrail
      Contact( #Ap_ET14 )
      wire#w2
      Contact( #PosicionConocida )
   END_RUNG wire#w1
   RUNG wire#powerrail
      Contact( #Ap_ET23 )
   END_RUNG wire#w2
   // the same network as SCL:
   #MA_Ir_Up := ((#Ap_ET104 AND NOT #MA_Ir_Dw) OR ((#Ap_ET14 OR #Ap_ET23) AND #PosicionConocida)) AND NOT #Pos_Up AND NOT #EM_UP AND NOT #EM_DW AND #EstadoZona.Marcha_CBx AND NOT #EstadoZona.Error_CBx AND NOT #EstadoZona.Error_CBx AND NOT #Error_Tx;
END_REGION

REGION Network 68: ESTADOS DE LA MAQUINA
   RUNG wire#powerrail
      Contact( TRUE )
      wire#w1
      Contact( #Ap_ET00 )
      Contact( #EstadoZona.PerReset_CBx )
      Coil( #EstadoMAQ.Etapa_Reset )
   END_RUNG
   RUNG wire#w1
      Contact( #STAT_Quieto )
      Coil( #EstadoMAQ.Etapa_EnReposo )
   END_RUNG
   RUNG wire#w1
      I_Contact( #STAT_Quieto )
      Coil( #EstadoMAQ.Etapa_EnMovimiento )
   END_RUNG
   // the same network as SCL:
   #EstadoMAQ.Etapa_Reset := TRUE AND #Ap_ET00 AND #EstadoZona.PerReset_CBx;
   #EstadoMAQ.Etapa_EnReposo := TRUE AND #STAT_Quieto;
   #EstadoMAQ.Etapa_EnMovimiento := TRUE AND NOT #STAT_Quieto;
END_REGION

REGION Network 69: ENTRADAS DE LA MAQUINA
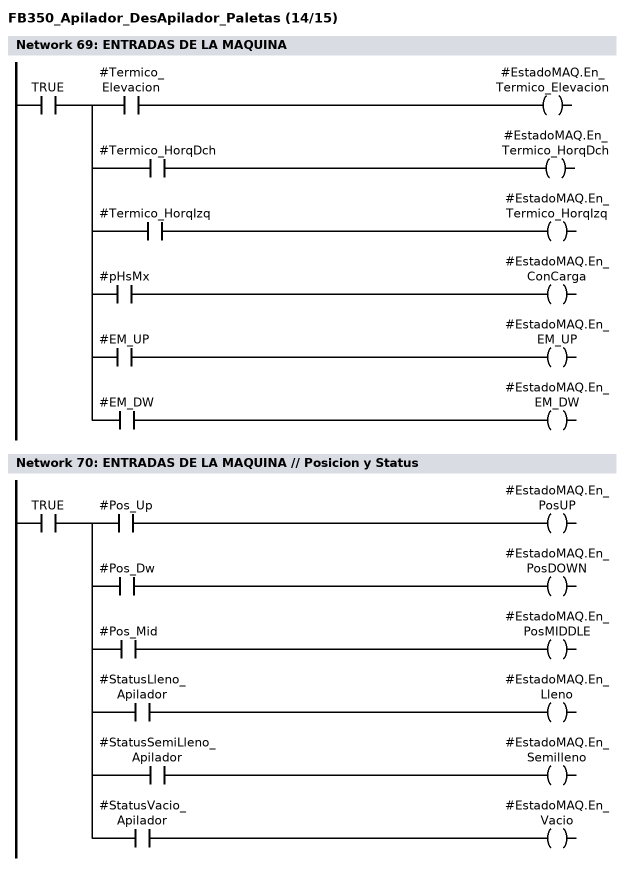
   RUNG wire#powerrail
      Contact( TRUE )
      wire#w1
      Contact( #Termico_Elevacion )
      Coil( #EstadoMAQ.En_Termico_Elevacion )
   END_RUNG
   RUNG wire#w1
      Contact( #Termico_HorqDch )
      Coil( #EstadoMAQ.En_Termico_HorqDch )
   END_RUNG
   RUNG wire#w1
      Contact( #Termico_HorqIzq )
      Coil( #EstadoMAQ.En_Termico_HorqIzq )
   END_RUNG
   RUNG wire#w1
      Contact( #pHsMx )
      Coil( #EstadoMAQ.En_ConCarga )
   END_RUNG
   RUNG wire#w1
      Contact( #EM_UP )
      Coil( #EstadoMAQ.En_EM_UP )
   END_RUNG
   RUNG wire#w1
      Contact( #EM_DW )
      Coil( #EstadoMAQ.En_EM_DW )
   END_RUNG
   // the same network as SCL:
   #EstadoMAQ.En_Termico_Elevacion := TRUE AND #Termico_Elevacion;
   #EstadoMAQ.En_Termico_HorqDch := TRUE AND #Termico_HorqDch;
   #EstadoMAQ.En_Termico_HorqIzq := TRUE AND #Termico_HorqIzq;
   #EstadoMAQ.En_ConCarga := TRUE AND #pHsMx;
   #EstadoMAQ.En_EM_UP := TRUE AND #EM_UP;
   #EstadoMAQ.En_EM_DW := TRUE AND #EM_DW;
END_REGION

REGION Network 70: ENTRADAS DE LA MAQUINA // Posicion y Status
   RUNG wire#powerrail
      Contact( TRUE )
      wire#w1
      Contact( #Pos_Up )
      Coil( #EstadoMAQ.En_PosUP )
   END_RUNG
   RUNG wire#w1
      Contact( #Pos_Dw )
      Coil( #EstadoMAQ.En_PosDOWN )
   END_RUNG
   RUNG wire#w1
      Contact( #Pos_Mid )
      Coil( #EstadoMAQ.En_PosMIDDLE )
   END_RUNG
   RUNG wire#w1
      Contact( #StatusLleno_Apilador )
      Coil( #EstadoMAQ.En_Lleno )
   END_RUNG
   RUNG wire#w1
      Contact( #StatusSemiLleno_Apilador )
      Coil( #EstadoMAQ.En_Semilleno )
   END_RUNG
   RUNG wire#w1
      Contact( #StatusVacio_Apilador )
      Coil( #EstadoMAQ.En_Vacio )
   END_RUNG
   // the same network as SCL:
   #EstadoMAQ.En_PosUP := TRUE AND #Pos_Up;
   #EstadoMAQ.En_PosDOWN := TRUE AND #Pos_Dw;
   #EstadoMAQ.En_PosMIDDLE := TRUE AND #Pos_Mid;
   #EstadoMAQ.En_Lleno := TRUE AND #StatusLleno_Apilador;
   #EstadoMAQ.En_Semilleno := TRUE AND #StatusSemiLleno_Apilador;
   #EstadoMAQ.En_Vacio := TRUE AND #StatusVacio_Apilador;
END_REGION

REGION Network 71: ENTRADAS DE LA MAQUINA // Sensores de las horquillas
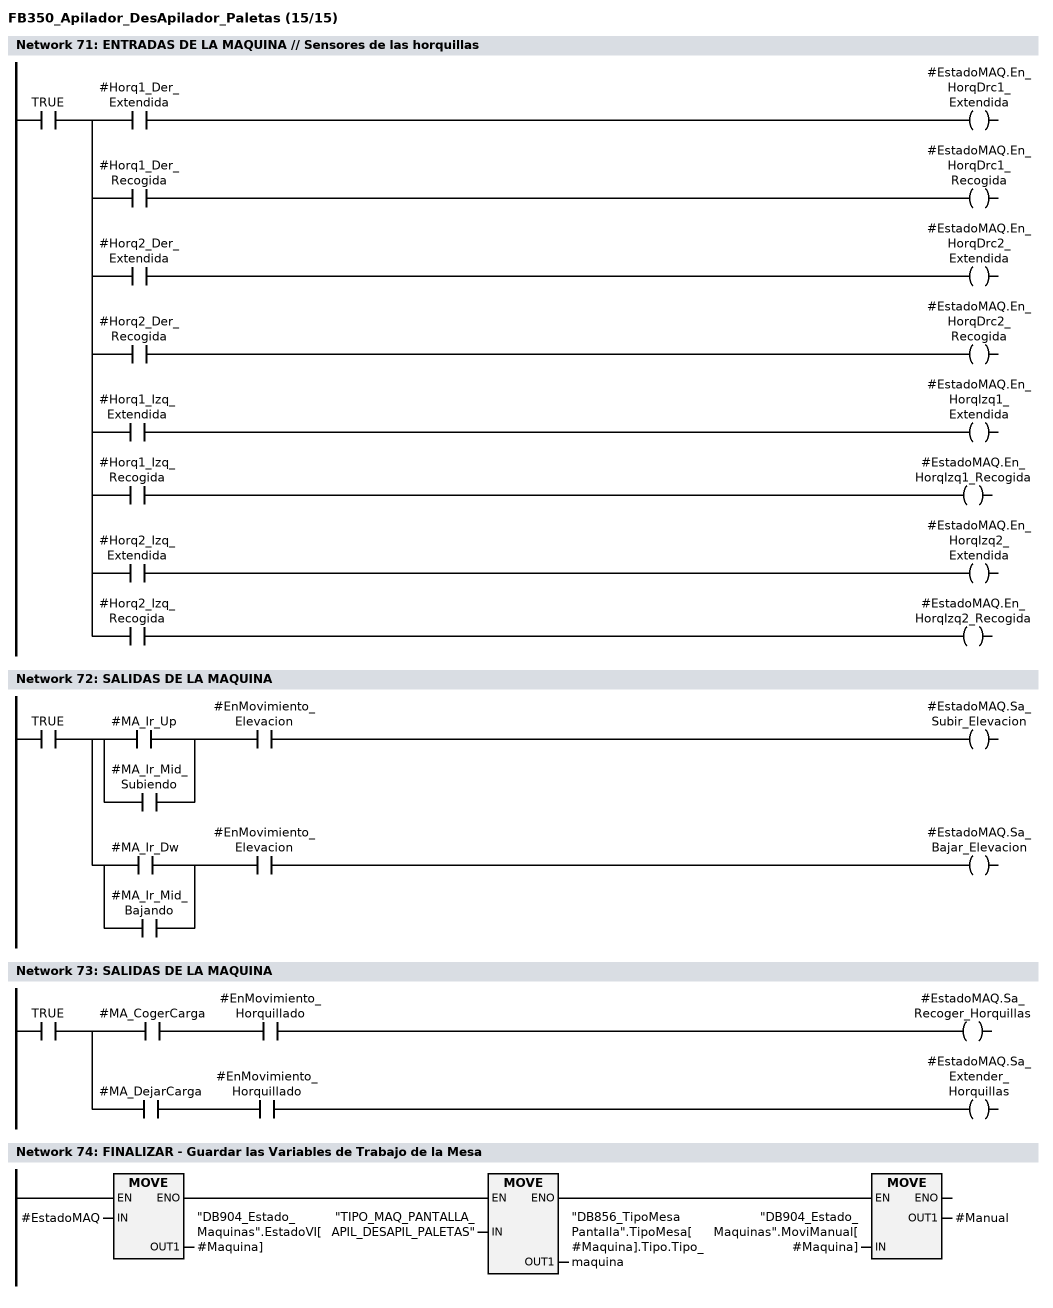
   RUNG wire#powerrail
      Contact( TRUE )
      wire#w1
      Contact( #Horq1_Der_Extendida )
      Coil( #EstadoMAQ.En_HorqDrc1_Extendida )
   END_RUNG
   RUNG wire#w1
      Contact( #Horq1_Der_Recogida )
      Coil( #EstadoMAQ.En_HorqDrc1_Recogida )
   END_RUNG
   RUNG wire#w1
      Contact( #Horq2_Der_Extendida )
      Coil( #EstadoMAQ.En_HorqDrc2_Extendida )
   END_RUNG
   RUNG wire#w1
      Contact( #Horq2_Der_Recogida )
      Coil( #EstadoMAQ.En_HorqDrc2_Recogida )
   END_RUNG
   RUNG wire#w1
      Contact( #Horq1_Izq_Extendida )
      Coil( #EstadoMAQ.En_HorqIzq1_Extendida )
   END_RUNG
   RUNG wire#w1
      Contact( #Horq1_Izq_Recogida )
      Coil( #EstadoMAQ.En_HorqIzq1_Recogida )
   END_RUNG
   RUNG wire#w1
      Contact( #Horq2_Izq_Extendida )
      Coil( #EstadoMAQ.En_HorqIzq2_Extendida )
   END_RUNG
   RUNG wire#w1
      Contact( #Horq2_Izq_Recogida )
      Coil( #EstadoMAQ.En_HorqIzq2_Recogida )
   END_RUNG
   // the same network as SCL:
   #EstadoMAQ.En_HorqDrc1_Extendida := TRUE AND #Horq1_Der_Extendida;
   #EstadoMAQ.En_HorqDrc1_Recogida := TRUE AND #Horq1_Der_Recogida;
   #EstadoMAQ.En_HorqDrc2_Extendida := TRUE AND #Horq2_Der_Extendida;
   #EstadoMAQ.En_HorqDrc2_Recogida := TRUE AND #Horq2_Der_Recogida;
   #EstadoMAQ.En_HorqIzq1_Extendida := TRUE AND #Horq1_Izq_Extendida;
   #EstadoMAQ.En_HorqIzq1_Recogida := TRUE AND #Horq1_Izq_Recogida;
   #EstadoMAQ.En_HorqIzq2_Extendida := TRUE AND #Horq2_Izq_Extendida;
   #EstadoMAQ.En_HorqIzq2_Recogida := TRUE AND #Horq2_Izq_Recogida;
END_REGION

REGION Network 72: SALIDAS DE LA MAQUINA
   RUNG wire#powerrail
      Contact( TRUE )
      wire#w1
      Contact( #MA_Ir_Up )
      wire#w2
      Contact( #EnMovimiento_Elevacion )
      Coil( #EstadoMAQ.Sa_Subir_Elevacion )
   END_RUNG
   RUNG wire#w1
      Contact( #MA_Ir_Mid_Subiendo )
   END_RUNG wire#w2
   RUNG wire#w1
      Contact( #MA_Ir_Dw )
      wire#w3
      Contact( #EnMovimiento_Elevacion )
      Coil( #EstadoMAQ.Sa_Bajar_Elevacion )
   END_RUNG
   RUNG wire#w1
      Contact( #MA_Ir_Mid_Bajando )
   END_RUNG wire#w3
   // the same network as SCL:
   #EstadoMAQ.Sa_Subir_Elevacion := TRUE AND (#MA_Ir_Up OR #MA_Ir_Mid_Subiendo) AND #EnMovimiento_Elevacion;
   #EstadoMAQ.Sa_Bajar_Elevacion := TRUE AND (#MA_Ir_Dw OR #MA_Ir_Mid_Bajando) AND #EnMovimiento_Elevacion;
END_REGION

REGION Network 73: SALIDAS DE LA MAQUINA
   RUNG wire#powerrail
      Contact( TRUE )
      wire#w1
      Contact( #MA_CogerCarga )
      Contact( #EnMovimiento_Horquillado )
      Coil( #EstadoMAQ.Sa_Recoger_Horquillas )
   END_RUNG
   RUNG wire#w1
      Contact( #MA_DejarCarga )
      Contact( #EnMovimiento_Horquillado )
      Coil( #EstadoMAQ.Sa_Extender_Horquillas )
   END_RUNG
   // the same network as SCL:
   #EstadoMAQ.Sa_Recoger_Horquillas := TRUE AND #MA_CogerCarga AND #EnMovimiento_Horquillado;
   #EstadoMAQ.Sa_Extender_Horquillas := TRUE AND #MA_DejarCarga AND #EnMovimiento_Horquillado;
END_REGION

REGION Network 74: FINALIZAR - Guardar las Variables de Trabajo de la Mesa
   RUNG wire#powerrail
      Move(in := #EstadoMAQ, out1 => "DB904_Estado_Maquinas".EstadoVI[#Maquina])
      Move(in := "TIPO_MAQ_PANTALLA_APIL_DESAPIL_PALETAS", out1 => "DB856_TipoMesaPantalla".TipoMesa[#Maquina].Tipo.Tipo_maquina)
      Move(in := "DB904_Estado_Maquinas".MoviManual[#Maquina], out1 => #Manual)
   END_RUNG
   // the same network as SCL:
   "DB904_Estado_Maquinas".EstadoVI[#Maquina] := #EstadoMAQ;
   "DB856_TipoMesaPantalla".TipoMesa[#Maquina].Tipo.Tipo_maquina := "TIPO_MAQ_PANTALLA_APIL_DESAPIL_PALETAS";
   #Manual := "DB904_Estado_Maquinas".MoviManual[#Maquina];
END_REGION
END_FUNCTION_BLOCK
